legal notes
=================
| SPDX-FileCopyrightText: © 2022 ekvip automation GmbH <info@ekvip.de>
| SPDX-License-Identifier: Apache-2.0
| For details check: Apache-2.0_

.. _Apache-2.0: https://www.apache.org/licenses/LICENSE-2.0

.. </legal notes>

parameters
=================

*)

METHOD bitXIsSet
VAR_INPUT
	(* current value to check *)
	currentValue	:__XWORD;
	(* number of bit to check *)
	number			:BitNumberXWord;	
	(* message if the assertion is false *)
	message			:AssertMessage;
END_VAR
END_METHOD

(*

short summary
=================
This assertion method checks if the selected bit of current value
is unset

.. <legal notes>

legal notes
=================
| SPDX-FileCopyrightText: © 2022 ekvip automation GmbH <info@ekvip.de>
| SPDX-License-Identifier: Apache-2.0
| For details check: Apache-2.0_

.. _Apache-2.0: https://www.apache.org/licenses/LICENSE-2.0

.. </legal notes>

parameters
=================

*)

METHOD bitXIsUnset
VAR_INPUT
	(* current value to check *)
	currentValue	:__XWORD;
	(* number of bit to check *)
	number			:BitNumberXWord;	
	(* message if the assertion is false *)
	message			:AssertMessage;
END_VAR
END_METHOD

(*

short summary
=================
This assertion method checks if the least significant bit of current value
is equal to the expected value

.. <legal notes>

legal notes
=================
| SPDX-FileCopyrightText: © 2022 ekvip automation GmbH <info@ekvip.de>
| SPDX-License-Identifier: Apache-2.0
| For details check: Apache-2.0_

.. _Apache-2.0: https://www.apache.org/licenses/LICENSE-2.0

.. </legal notes>

parameters
=================

*)

METHOD lsbIsEqualTo
VAR_INPUT
	(* current value to check *)
	currentValue	:__XWORD;
	(* expected value of lsb *)
	expectedValue	:BOOL;
	(* message if the assertion is false *)
	message			:AssertMessage;
END_VAR
END_METHOD

(*

short summary
=================
This assertion method checks if the least significant bit of current value
is not equal to the unexpected value

.. <legal notes>

legal notes
=================
| SPDX-FileCopyrightText: © 2022 ekvip automation GmbH <info@ekvip.de>
| SPDX-License-Identifier: Apache-2.0
| For details check: Apache-2.0_

.. _Apache-2.0: https://www.apache.org/licenses/LICENSE-2.0

.. </legal notes>

parameters
=================

*)

METHOD lsbIsNotEqualTo
VAR_INPUT
	(* current value to check *)
	currentValue	:__XWORD;
	(* unexpected value of lsb *)
	unexpectedValue	:BOOL;
	(* message if the assertion is false *)
	message			:AssertMessage;
END_VAR
END_METHOD

(*

short summary
=================
This assertion method checks if the least significant bit of current value
is set

.. <legal notes>

legal notes
=================
| SPDX-FileCopyrightText: © 2022 ekvip automation GmbH <info@ekvip.de>
| SPDX-License-Identifier: Apache-2.0
| For details check: Apache-2.0_

.. _Apache-2.0: https://www.apache.org/licenses/LICENSE-2.0

.. </legal notes>

parameters
=================

*)

METHOD lsbIsSet
VAR_INPUT
	(* current value to check *)
	currentValue	:__XWORD;
	(* message if the assertion is false *)
	message			:AssertMessage;
END_VAR
END_METHOD

(*

short summary
=================
This assertion method checks if the least significant bit of current value
is unset

.. <legal notes>

legal notes
=================
| SPDX-FileCopyrightText: © 2022 ekvip automation GmbH <info@ekvip.de>
| SPDX-License-Identifier: Apache-2.0
| For details check: Apache-2.0_

.. _Apache-2.0: https://www.apache.org/licenses/LICENSE-2.0

.. </legal notes>

parameters
=================

*)

METHOD lsbIsUnset
VAR_INPUT
	(* current value to check *)
	currentValue	:__XWORD;
	(* message if the assertion is false *)
	message			:AssertMessage;
END_VAR
END_METHOD

(*

short summary
=================
This assertion method checks if the most significant bit of current value
is equal to the expected value

.. <legal notes>

legal notes
=================
| SPDX-FileCopyrightText: © 2022 ekvip automation GmbH <info@ekvip.de>
| SPDX-License-Identifier: Apache-2.0
| For details check: Apache-2.0_

.. _Apache-2.0: https://www.apache.org/licenses/LICENSE-2.0

.. </legal notes>

parameters
=================

*)

METHOD msbIsEqualTo
VAR_INPUT
	(* current value to check *)
	currentValue	:__XWORD;
	(* expected value of msb *)
	expectedValue	:BOOL;
	(* message if the assertion is false *)
	message			:AssertMessage;
END_VAR
END_METHOD

(*

short summary
=================
This assertion method checks if the most significant bit of current value
is not equal to the unexpected value

.. <legal notes>

legal notes
=================
| SPDX-FileCopyrightText: © 2022 ekvip automation GmbH <info@ekvip.de>
| SPDX-License-Identifier: Apache-2.0
| For details check: Apache-2.0_

.. _Apache-2.0: https://www.apache.org/licenses/LICENSE-2.0

.. </legal notes>

parameters
=================

*)

METHOD msbIsNotEqualTo
VAR_INPUT
	(* current value to check *)
	currentValue	:__XWORD;
	(* unexpected value of msb *)
	unexpectedValue	:BOOL;
	(* message if the assertion is false *)
	message			:AssertMessage;
END_VAR
END_METHOD

(*

short summary
=================
This assertion method checks if the most significant bit of current value
is set

.. <legal notes>

legal notes
=================
| SPDX-FileCopyrightText: © 2022 ekvip automation GmbH <info@ekvip.de>
| SPDX-License-Identifier: Apache-2.0
| For details check: Apache-2.0_

.. _Apache-2.0: https://www.apache.org/licenses/LICENSE-2.0

.. </legal notes>

parameters
=================

*)

METHOD msbIsSet
VAR_INPUT
	(* current value to check *)
	currentValue	:__XWORD;
	(* message if the assertion is false *)
	message			:AssertMessage;
END_VAR
END_METHOD

(*

short summary
=================
This assertion method checks if the most significant bit of current value
is unset

.. <legal notes>

legal notes
=================
| SPDX-FileCopyrightText: © 2022 ekvip automation GmbH <info@ekvip.de>
| SPDX-License-Identifier: Apache-2.0
| For details check: Apache-2.0_

.. _Apache-2.0: https://www.apache.org/licenses/LICENSE-2.0

.. </legal notes>

parameters
=================

*)

METHOD msbIsUnset
VAR_INPUT
	(* current value to check *)
	currentValue	:__XWORD;
	(* message if the assertion is false *)
	message			:AssertMessage;
END_VAR
END_METHOD

(*

short summary
=================
This assertion method checks if the result current value bitwise ``OR`` mask is equal to the expected value

.. <legal notes>

legal notes
=================
| SPDX-FileCopyrightText: © 2022 ekvip automation GmbH <info@ekvip.de>
| SPDX-License-Identifier: Apache-2.0
| For details check: Apache-2.0_

.. _Apache-2.0: https://www.apache.org/licenses/LICENSE-2.0

.. </legal notes>

parameters
=================

*)

METHOD orMaskIsEqualTo
VAR_INPUT
	(* current value to check *)
	currentValue	:__XWORD;
	(* 2nd operand for bitwise operation *)
	mask			:__XWORD;
	(* expected result after masking *)
	expectedValue	:__XWORD;
	(* message if the assertion is false *)
	message			:AssertMessage;
END_VAR
END_METHOD

(*

short summary
=================
This assertion method checks if the result current value bitwise ``OR`` mask 
is not equal to the unexpected value

.. <legal notes>

legal notes
=================
| SPDX-FileCopyrightText: © 2022 ekvip automation GmbH <info@ekvip.de>
| SPDX-License-Identifier: Apache-2.0
| For details check: Apache-2.0_

.. _Apache-2.0: https://www.apache.org/licenses/LICENSE-2.0

.. </legal notes>

parameters
=================

*)

METHOD orMaskIsNotEqualTo
VAR_INPUT
	(* current value to check *)
	currentValue	:__XWORD;
	(* 2nd operand for bitwise operation *)
	mask			:__XWORD;
	(* unexpected result after masking *)
	unexpectedValue	:__XWORD;
	(* message if the assertion is false *)
	message			:AssertMessage;
END_VAR
END_METHOD

(*

short summary
=================
This assertion method checks if the current value is equal to the expected value

.. <legal notes>

legal notes
=================
| SPDX-FileCopyrightText: © 2022 ekvip automation GmbH <info@ekvip.de>
| SPDX-License-Identifier: Apache-2.0
| For details check: Apache-2.0_

.. _Apache-2.0: https://www.apache.org/licenses/LICENSE-2.0

.. </legal notes>

parameters
=================

*)

METHOD valueIsEqualTo
VAR_INPUT
	(* current value to check *)
	currentValue	:__XWORD;
	(* expected value to compare *)
	expectedValue	:__XWORD;
	(* message if the assertion is false *)
	message			:AssertMessage;
END_VAR
END_METHOD

(*

short summary
=================
This assertion method checks if the current value is greater than the less value

.. <legal notes>

legal notes
=================
| SPDX-FileCopyrightText: © 2022 ekvip automation GmbH <info@ekvip.de>
| SPDX-License-Identifier: Apache-2.0
| For details check: Apache-2.0_

.. _Apache-2.0: https://www.apache.org/licenses/LICENSE-2.0

.. </legal notes>

parameters
=================

*)

METHOD valueIsGreaterThan
VAR_INPUT
	(* current value to check *)
	currentValue	:__XWORD;
	(* less than lower limit *)
	lessValue		:__XWORD;
	(* message if the assertion is false *)
	message			:AssertMessage;
END_VAR
END_METHOD

(*

short summary
=================
This assertion method checks if the current value is inside a limit

.. attention:: 
	limits are included: ``valueIsInRangeOf(3, 3, 3)`` is a true assertion

.. <legal notes>

legal notes
=================
| SPDX-FileCopyrightText: © 2022 ekvip automation GmbH <info@ekvip.de>
| SPDX-License-Identifier: Apache-2.0
| For details check: Apache-2.0_

.. _Apache-2.0: https://www.apache.org/licenses/LICENSE-2.0

.. </legal notes>

parameters
=================

*)

METHOD valueIsInRangeOf
VAR_INPUT
	(* lower limit for the current value *)
	lowerLimit		:__XWORD;
	(* current value to check *)
	currentValue	:__XWORD;
	(* upper limit for the current value *)
	upperLimit		:__XWORD;
	(* message if the assertion is false *)
	message			:AssertMessage;
END_VAR
END_METHOD

(*

short summary
=================
This assertion method checks if the current value is less than the greater value

.. <legal notes>

legal notes
=================
| SPDX-FileCopyrightText: © 2022 ekvip automation GmbH <info@ekvip.de>
| SPDX-License-Identifier: Apache-2.0
| For details check: Apache-2.0_

.. _Apache-2.0: https://www.apache.org/licenses/LICENSE-2.0

.. </legal notes>

parameters
=================

*)

METHOD valueIsLessThan
VAR_INPUT
	(* current value to check *)
	currentValue	:__XWORD;
	(* greater than upper limit *)
	greaterValue	:__XWORD;
	(* message if the assertion is false *)
	message			:AssertMessage;
END_VAR
END_METHOD

(*

short summary
=================
This assertion method checks if the current value is less than or equal to the maximum value

.. <legal notes>

legal notes
=================
| SPDX-FileCopyrightText: © 2022 ekvip automation GmbH <info@ekvip.de>
| SPDX-License-Identifier: Apache-2.0
| For details check: Apache-2.0_

.. _Apache-2.0: https://www.apache.org/licenses/LICENSE-2.0

.. </legal notes>

parameters
=================

*)

METHOD valueIsMax
VAR_INPUT
	(* current value to check *)
	currentValue	:__XWORD;
	(* upper limit for the current value *)
	maximumValue	:__XWORD;
	(* message if the assertion is false *)
	message			:AssertMessage;
END_VAR
END_METHOD

(*

short summary
=================
This assertion method checks if the current value is greater than or equal to the minimum value

.. <legal notes>

legal notes
=================
| SPDX-FileCopyrightText: © 2022 ekvip automation GmbH <info@ekvip.de>
| SPDX-License-Identifier: Apache-2.0
| For details check: Apache-2.0_

.. _Apache-2.0: https://www.apache.org/licenses/LICENSE-2.0

.. </legal notes>

parameters
=================

*)

METHOD valueIsMin
VAR_INPUT
	(* current value to check *)
	currentValue	:__XWORD;
	(* lower limit for the current value *)
	minimumValue	:__XWORD;
	(* message if the assertion is false *)
	message			:AssertMessage;
END_VAR
END_METHOD

(*

short summary
=================
This assertion method checks if the current value is not equal to the unexpected value

.. <legal notes>

legal notes
=================
| SPDX-FileCopyrightText: © 2022 ekvip automation GmbH <info@ekvip.de>
| SPDX-License-Identifier: Apache-2.0
| For details check: Apache-2.0_

.. _Apache-2.0: https://www.apache.org/licenses/LICENSE-2.0

.. </legal notes>

parameters
=================

*)

METHOD valueIsNotEqualTo
VAR_INPUT
	(* current value to check *)
	currentValue	:__XWORD;
	(* unexpected value to compare *)
	unexpectedValue	:__XWORD;
	(* message if the assertion is false *)
	message			:AssertMessage;
END_VAR
END_METHOD

(*

short summary
=================
This assertion method checks if the result current value bitwise ``XOR`` mask is equal to the expected value

.. <legal notes>

legal notes
=================
| SPDX-FileCopyrightText: © 2022 ekvip automation GmbH <info@ekvip.de>
| SPDX-License-Identifier: Apache-2.0
| For details check: Apache-2.0_

.. _Apache-2.0: https://www.apache.org/licenses/LICENSE-2.0

.. </legal notes>

parameters
=================

*)

METHOD xorMaskIsEqualTo
VAR_INPUT
	(* current value to check *)
	currentValue	:__XWORD;
	(* 2nd operand for bitwise operation *)
	mask			:__XWORD;
	(* expected result after masking *)
	expectedValue	:__XWORD;
	(* message if the assertion is false *)
	message			:AssertMessage;
END_VAR
END_METHOD

(*

short summary
=================
This assertion method checks if the result current value bitwise ``XOR`` mask 
is not equal to the unexpected value

.. <legal notes>

legal notes
=================
| SPDX-FileCopyrightText: © 2022 ekvip automation GmbH <info@ekvip.de>
| SPDX-License-Identifier: Apache-2.0
| For details check: Apache-2.0_

.. _Apache-2.0: https://www.apache.org/licenses/LICENSE-2.0

.. </legal notes>

parameters
=================

*)

METHOD xorMaskIsNotEqualTo
VAR_INPUT
	(* current value to check *)
	currentValue	:__XWORD;
	(* 2nd operand for bitwise operation *)
	mask			:__XWORD;
	(* unexpected result after masking *)
	unexpectedValue	:__XWORD;
	(* message if the assertion is false *)
	message			:AssertMessage;
END_VAR
END_METHOD

END_INTERFACE

// ---- Assertor/Assertions/BooleanAssertion/interfaces/IBooleanAssertion.TcIO
(*

short summary
=================
This interface provides assert statements for booleans 

.. <legal notes>

legal notes
=================
| SPDX-FileCopyrightText: © 2022 ekvip automation GmbH <info@ekvip.de>
| SPDX-License-Identifier: Apache-2.0
| For details check: Apache-2.0_

.. _Apache-2.0: https://www.apache.org/licenses/LICENSE-2.0

.. </legal notes>

methods
==================

*)

INTERFACE IBooleanAssertion EXTENDS __SYSTEM.IQueryInterface

(*

short summary
=================
This assertion method checks if the current value is equal to the expected value

.. <legal notes>

legal notes
=================
| SPDX-FileCopyrightText: © 2022 ekvip automation GmbH <info@ekvip.de>
| SPDX-License-Identifier: Apache-2.0
| For details check: Apache-2.0_

.. _Apache-2.0: https://www.apache.org/licenses/LICENSE-2.0

.. </legal notes>

parameters
=================

*)

METHOD valueIsEqualTo
VAR_INPUT
	(* current value to check *)
	currentValue	:BOOL;
	(* expected value to compare *)
	expectedValue	:BOOL;
	(* message if the assertion is false *)
	message			:AssertMessage;
END_VAR
END_METHOD

(*

short summary
=================
This assertion method checks if the current value is ``FALSE``

.. <legal notes>

legal notes
=================
| SPDX-FileCopyrightText: © 2022 ekvip automation GmbH <info@ekvip.de>
| SPDX-License-Identifier: Apache-2.0
| For details check: Apache-2.0_

.. _Apache-2.0: https://www.apache.org/licenses/LICENSE-2.0

.. </legal notes>

parameters
=================

*)

METHOD valueIsFalse
VAR_INPUT
	(* current value to check *)
	currentValue	:BOOL;
	(* message if the assertion is false *)
	message			:AssertMessage;
END_VAR
END_METHOD

(*

short summary
=================
This assertion method checks if the current value is not equal to the unexpected value

.. <legal notes>

legal notes
=================
| SPDX-FileCopyrightText: © 2022 ekvip automation GmbH <info@ekvip.de>
| SPDX-License-Identifier: Apache-2.0
| For details check: Apache-2.0_

.. _Apache-2.0: https://www.apache.org/licenses/LICENSE-2.0

.. </legal notes>

parameters
=================

*)

METHOD valueIsNotEqualTo
VAR_INPUT
	(* current value to check *)
	currentValue	:BOOL;
	(* unexpected value to compare *)
	unexpectedValue	:BOOL;
	(* message if the assertion is false *)
	message			:AssertMessage;
END_VAR
END_METHOD

(*

short summary
=================
This assertion method checks if the current value is ``TRUE``

.. <legal notes>

legal notes
=================
| SPDX-FileCopyrightText: © 2022 ekvip automation GmbH <info@ekvip.de>
| SPDX-License-Identifier: Apache-2.0
| For details check: Apache-2.0_

.. _Apache-2.0: https://www.apache.org/licenses/LICENSE-2.0

.. </legal notes>

parameters
=================

*)

METHOD valueIsTrue
VAR_INPUT
	(* current value to check *)
	currentValue	:BOOL;
	(* message if the assertion is false *)
	message			:AssertMessage;
END_VAR
END_METHOD

END_INTERFACE

// ---- Assertor/Assertions/DateAndTimeAssertions/32Bit/Date/interfaces/I32BitDateAssertions.TcIO
(*

short summary
=================
This interface provides assert statements for 32 bit ``DATE``  

.. <legal notes>

legal notes
=================
| SPDX-FileCopyrightText: © 2022 ekvip automation GmbH <info@ekvip.de>
| SPDX-License-Identifier: Apache-2.0
| For details check: Apache-2.0_

.. _Apache-2.0: https://www.apache.org/licenses/LICENSE-2.0

.. </legal notes>

methods
==================

*)

INTERFACE I32BitDateAssertions EXTENDS __SYSTEM.IQueryInterface

(*

short summary
=================
This assertion method checks if the current value is equal to the expected value

.. <legal notes>

legal notes
=================
| SPDX-FileCopyrightText: © 2022 ekvip automation GmbH <info@ekvip.de>
| SPDX-License-Identifier: Apache-2.0
| For details check: Apache-2.0_

.. _Apache-2.0: https://www.apache.org/licenses/LICENSE-2.0

.. </legal notes>

parameters
=================

*)

METHOD valueIsEqualTo
VAR_INPUT
	(* current value to check *)
	currentValue	:DATE;
	(* expected value to compare *)
	expectedValue	:DATE;
	(* message if the assertion is false *)
	message			:AssertMessage;
END_VAR
END_METHOD

(*

short summary
=================
This assertion method checks if the current value is greater than the less value

.. <legal notes>

legal notes
=================
| SPDX-FileCopyrightText: © 2022 ekvip automation GmbH <info@ekvip.de>
| SPDX-License-Identifier: Apache-2.0
| For details check: Apache-2.0_

.. _Apache-2.0: https://www.apache.org/licenses/LICENSE-2.0

.. </legal notes>

parameters
=================

*)

METHOD valueIsGreaterThan
VAR_INPUT
	(* current value to check *)
	currentValue	:DATE;
	(* less than lower limit *)
	lessValue		:DATE;
	(* message if the assertion is false *)
	message			:AssertMessage;
END_VAR
END_METHOD

(*

short summary
=================
This assertion method checks if the current value is inside a limit

.. attention:: 
	limits are included: ``valueIsInRangeOf(date#1970-01-01, date#1970-01-01, date#1970-01-01)``
	is a true assertion

.. <legal notes>

legal notes
=================
| SPDX-FileCopyrightText: © 2022 ekvip automation GmbH <info@ekvip.de>
| SPDX-License-Identifier: Apache-2.0
| For details check: Apache-2.0_

.. _Apache-2.0: https://www.apache.org/licenses/LICENSE-2.0

.. </legal notes>

parameters
=================

*)

METHOD valueIsInRangeOf
VAR_INPUT
	(* lower limit for the current value *)
	lowerLimit		:DATE;
	(* current value to check *)
	currentValue	:DATE;
	(* upper limit for the current value *)
	upperLimit		:DATE;
	(* message if the assertion is false *)
	message			:AssertMessage;
END_VAR
END_METHOD

(*

short summary
=================
This assertion method checks if the current value is less than the greater value

.. <legal notes>

legal notes
=================
| SPDX-FileCopyrightText: © 2022 ekvip automation GmbH <info@ekvip.de>
| SPDX-License-Identifier: Apache-2.0
| For details check: Apache-2.0_

.. _Apache-2.0: https://www.apache.org/licenses/LICENSE-2.0

.. </legal notes>

parameters
=================

*)

METHOD valueIsLessThan
VAR_INPUT
	(* current value to check *)
	currentValue	:DATE;
	(* greater than upper limit *)
	greaterValue	:DATE;
	(* message if the assertion is false *)
	message			:AssertMessage;
END_VAR
END_METHOD

(*

short summary
=================
This assertion method checks if the current value is less than or equal to the maximum value

.. <legal notes>

legal notes
=================
| SPDX-FileCopyrightText: © 2022 ekvip automation GmbH <info@ekvip.de>
| SPDX-License-Identifier: Apache-2.0
| For details check: Apache-2.0_

.. _Apache-2.0: https://www.apache.org/licenses/LICENSE-2.0

.. </legal notes>

parameters
=================

*)

METHOD valueIsMax
VAR_INPUT
	(* current value to check *)
	currentValue	:DATE;
	(* upper limit for the current value *)
	maximumValue	:DATE;
	(* message if the assertion is false *)
	message			:AssertMessage;
END_VAR
END_METHOD

(*

short summary
=================
This assertion method checks if the current value is greater than or equal to the minimum value

.. <legal notes>

legal notes
=================
| SPDX-FileCopyrightText: © 2022 ekvip automation GmbH <info@ekvip.de>
| SPDX-License-Identifier: Apache-2.0
| For details check: Apache-2.0_

.. _Apache-2.0: https://www.apache.org/licenses/LICENSE-2.0

.. </legal notes>

parameters
=================

*)

METHOD valueIsMin
VAR_INPUT
	(* current value to check *)
	currentValue	:DATE;
	(* lower limit for the current value *)
	minimumValue	:DATE;
	(* message if the assertion is false *)
	message			:AssertMessage;
END_VAR
END_METHOD

(*

short summary
=================
This assertion method checks if the current value is not equal to the unexpected value

.. <legal notes>

legal notes
=================
| SPDX-FileCopyrightText: © 2022 ekvip automation GmbH <info@ekvip.de>
| SPDX-License-Identifier: Apache-2.0
| For details check: Apache-2.0_

.. _Apache-2.0: https://www.apache.org/licenses/LICENSE-2.0

.. </legal notes>

parameters
=================

*)

METHOD valueIsNotEqualTo
VAR_INPUT
	(* current value to check *)
	currentValue	:DATE;
	(* unexpected value to compare *)
	unexpectedValue	:DATE;
	(* message if the assertion is false *)
	message			:AssertMessage;
END_VAR
END_METHOD

END_INTERFACE

// ---- Assertor/Assertions/DateAndTimeAssertions/32Bit/DT/interfaces/I32BitDtAssertions.TcIO
(*

short summary
=================
This interface provides assert statements for 32 bit date and time ``DT``  

.. <legal notes>

legal notes
=================
| SPDX-FileCopyrightText: © 2022 ekvip automation GmbH <info@ekvip.de>
| SPDX-License-Identifier: Apache-2.0
| For details check: Apache-2.0_

.. _Apache-2.0: https://www.apache.org/licenses/LICENSE-2.0

.. </legal notes>

methods
==================

*)

INTERFACE I32BitDtAssertions EXTENDS __SYSTEM.IQueryInterface

(*

short summary
=================
This assertion method checks if the current value is equal to the expected value

.. <legal notes>

legal notes
=================
| SPDX-FileCopyrightText: © 2022 ekvip automation GmbH <info@ekvip.de>
| SPDX-License-Identifier: Apache-2.0
| For details check: Apache-2.0_

.. _Apache-2.0: https://www.apache.org/licenses/LICENSE-2.0

.. </legal notes>

parameters
=================

*)

METHOD valueIsEqualTo
VAR_INPUT
	(* current value to check *)
	currentValue	:DT;
	(* expected value to compare *)
	expectedValue	:DT;
	(* message if the assertion is false *)
	message			:AssertMessage;
END_VAR
END_METHOD

(*

short summary
=================
This assertion method checks if the current value is greater than the less value

.. <legal notes>

legal notes
=================
| SPDX-FileCopyrightText: © 2022 ekvip automation GmbH <info@ekvip.de>
| SPDX-License-Identifier: Apache-2.0
| For details check: Apache-2.0_

.. _Apache-2.0: https://www.apache.org/licenses/LICENSE-2.0

.. </legal notes>

parameters
=================

*)

METHOD valueIsGreaterThan
VAR_INPUT
	(* current value to check *)
	currentValue	:DT;
	(* less than lower limit *)
	lessValue		:DT;
	(* message if the assertion is false *)
	message			:AssertMessage;
END_VAR
END_METHOD

(*

short summary
=================
This assertion method checks if the current value is inside a limit

.. attention:: 
	limits are included: ``valueIsInRangeOf(dt#1970-01-01-0:0:0, dt#1970-01-01-0:0:0, dt#1970-01-01-0:0:0)``
	is a true assertion

.. <legal notes>

legal notes
=================
| SPDX-FileCopyrightText: © 2022 ekvip automation GmbH <info@ekvip.de>
| SPDX-License-Identifier: Apache-2.0
| For details check: Apache-2.0_

.. _Apache-2.0: https://www.apache.org/licenses/LICENSE-2.0

.. </legal notes>

parameters
=================

*)

METHOD valueIsInRangeOf
VAR_INPUT
	(* lower limit for the current value *)
	lowerLimit		:DT;
	(* current value to check *)
	currentValue	:DT;
	(* upper limit for the current value *)
	upperLimit		:DT;
	(* message if the assertion is false *)
	message			:AssertMessage;
END_VAR
END_METHOD

(*

short summary
=================
This assertion method checks if the current value is less than the greater value

.. <legal notes>

legal notes
=================
| SPDX-FileCopyrightText: © 2022 ekvip automation GmbH <info@ekvip.de>
| SPDX-License-Identifier: Apache-2.0
| For details check: Apache-2.0_

.. _Apache-2.0: https://www.apache.org/licenses/LICENSE-2.0

.. </legal notes>

parameters
=================

*)

METHOD valueIsLessThan
VAR_INPUT
	(* current value to check *)
	currentValue	:DT;
	(* greater than upper limit *)
	greaterValue	:DT;
	(* message if the assertion is false *)
	message			:AssertMessage;
END_VAR
END_METHOD

(*

short summary
=================
This assertion method checks if the current value is less than or equal to the maximum value

.. <legal notes>

legal notes
=================
| SPDX-FileCopyrightText: © 2022 ekvip automation GmbH <info@ekvip.de>
| SPDX-License-Identifier: Apache-2.0
| For details check: Apache-2.0_

.. _Apache-2.0: https://www.apache.org/licenses/LICENSE-2.0

.. </legal notes>

parameters
=================

*)

METHOD valueIsMax
VAR_INPUT
	(* current value to check *)
	currentValue	:DT;
	(* upper limit for the current value *)
	maximumValue	:DT;
	(* message if the assertion is false *)
	message			:AssertMessage;
END_VAR
END_METHOD

(*

short summary
=================
This assertion method checks if the current value is greater than or equal to the minimum value

.. <legal notes>

legal notes
=================
| SPDX-FileCopyrightText: © 2022 ekvip automation GmbH <info@ekvip.de>
| SPDX-License-Identifier: Apache-2.0
| For details check: Apache-2.0_

.. _Apache-2.0: https://www.apache.org/licenses/LICENSE-2.0

.. </legal notes>

parameters
=================

*)

METHOD valueIsMin
VAR_INPUT
	(* current value to check *)
	currentValue	:DT;
	(* lower limit for the current value *)
	minimumValue	:DT;
	(* message if the assertion is false *)
	message			:AssertMessage;
END_VAR
END_METHOD

(*

short summary
=================
This assertion method checks if the current value is not equal to the unexpected value

.. <legal notes>

legal notes
=================
| SPDX-FileCopyrightText: © 2022 ekvip automation GmbH <info@ekvip.de>
| SPDX-License-Identifier: Apache-2.0
| For details check: Apache-2.0_

.. _Apache-2.0: https://www.apache.org/licenses/LICENSE-2.0

.. </legal notes>

parameters
=================

*)

METHOD valueIsNotEqualTo
VAR_INPUT
	(* current value to check *)
	currentValue	:DT;
	(* unexpected value to compare *)
	unexpectedValue	:DT;
	(* message if the assertion is false *)
	message			:AssertMessage;
END_VAR
END_METHOD

END_INTERFACE

// ---- Assertor/Assertions/DateAndTimeAssertions/32Bit/interfaces/ISimpleDateAndTimeAssertions.TcIO
(*

short summary
=================
| This interface provides assert statements for date and time types with 32 bit length
| For date and time (``DT``) use :ref:`ISimpleDateAndTimeAssertions.dateAndTime`
| For date (``DATE``) use  :ref:`ISimpleDateAndTimeAssertions.dateOnly`
| For time of day (``TOD``) use  :ref:`ISimpleDateAndTimeAssertions.timeOfDay`

.. <legal notes>

legal notes
=================
| SPDX-FileCopyrightText: © 2022 ekvip automation GmbH <info@ekvip.de>
| SPDX-License-Identifier: Apache-2.0
| For details check: Apache-2.0_

.. _Apache-2.0: https://www.apache.org/licenses/LICENSE-2.0

.. </legal notes>

methods
==================

*)

INTERFACE ISimpleDateAndTimeAssertions EXTENDS __SYSTEM.IQueryInterface

(*

short summary
=================
Returns the interface :ref:`I32BitDtAssertions` with assert statements for 32 bit date and time ``DT``

.. <legal notes>

legal notes
=================
| SPDX-FileCopyrightText: © 2022 ekvip automation GmbH <info@ekvip.de>
| SPDX-License-Identifier: Apache-2.0
| For details check: Apache-2.0_

.. _Apache-2.0: https://www.apache.org/licenses/LICENSE-2.0

.. </legal notes>

*)

PROPERTY dateAndTime :I32BitDtAssertions
GET
END_GET
END_PROPERTY

(*

short summary
=================
Returns the interface :ref:`I32BitDateAssertions` with assert statements for 32 bit date ``DATE``

.. <legal notes>

legal notes
=================
| SPDX-FileCopyrightText: © 2022 ekvip automation GmbH <info@ekvip.de>
| SPDX-License-Identifier: Apache-2.0
| For details check: Apache-2.0_

.. _Apache-2.0: https://www.apache.org/licenses/LICENSE-2.0

.. </legal notes>

*)

PROPERTY dateOnly :I32BitDateAssertions
GET
END_GET
END_PROPERTY

(*

short summary
=================
Returns the interface :ref:`I32BitTodAssertions` with assert statements for 32 bit time of day ``TOD``

.. <legal notes>

legal notes
=================
| SPDX-FileCopyrightText: © 2022 ekvip automation GmbH <info@ekvip.de>
| SPDX-License-Identifier: Apache-2.0
| For details check: Apache-2.0_

.. _Apache-2.0: https://www.apache.org/licenses/LICENSE-2.0

.. </legal notes>

*)

PROPERTY timeOfDay :I32BitTodAssertions
GET
END_GET
END_PROPERTY

END_INTERFACE

// ---- Assertor/Assertions/DateAndTimeAssertions/32Bit/TOD/interfaces/I32BitTodAssertions.TcIO
(*

short summary
=================
This interface provides assert statements for 32 bit time of day ``TOD``  

.. <legal notes>

legal notes
=================
| SPDX-FileCopyrightText: © 2022 ekvip automation GmbH <info@ekvip.de>
| SPDX-License-Identifier: Apache-2.0
| For details check: Apache-2.0_

.. _Apache-2.0: https://www.apache.org/licenses/LICENSE-2.0

.. </legal notes>

methods
==================

*)

INTERFACE I32BitTodAssertions EXTENDS __SYSTEM.IQueryInterface

(*

short summary
=================
This assertion method checks if the current value is equal to the expected value

.. <legal notes>

legal notes
=================
| SPDX-FileCopyrightText: © 2022 ekvip automation GmbH <info@ekvip.de>
| SPDX-License-Identifier: Apache-2.0
| For details check: Apache-2.0_

.. _Apache-2.0: https://www.apache.org/licenses/LICENSE-2.0

.. </legal notes>

parameters
=================

*)

METHOD valueIsEqualTo
VAR_INPUT
	(* current value to check *)
	currentValue	:TOD;
	(* expected value to compare *)
	expectedValue	:TOD;
	(* message if the assertion is false *)
	message			:AssertMessage;
END_VAR
END_METHOD

(*

short summary
=================
This assertion method checks if the current value is greater than the less value

.. <legal notes>

legal notes
=================
| SPDX-FileCopyrightText: © 2022 ekvip automation GmbH <info@ekvip.de>
| SPDX-License-Identifier: Apache-2.0
| For details check: Apache-2.0_

.. _Apache-2.0: https://www.apache.org/licenses/LICENSE-2.0

.. </legal notes>

parameters
=================

*)

METHOD valueIsGreaterThan
VAR_INPUT
	(* current value to check *)
	currentValue	:TOD;
	(* less than lower limit *)
	lessValue		:TOD;
	(* message if the assertion is false *)
	message			:AssertMessage;
END_VAR
END_METHOD

(*

short summary
=================
This assertion method checks if the current value is inside a limit

.. attention:: 
	limits are included: ``valueIsInRangeOf(tod#3:0:0, tod#3:0:0, tod#3:0:0)`` is a true assertion

.. <legal notes>

legal notes
=================
| SPDX-FileCopyrightText: © 2022 ekvip automation GmbH <info@ekvip.de>
| SPDX-License-Identifier: Apache-2.0
| For details check: Apache-2.0_

.. _Apache-2.0: https://www.apache.org/licenses/LICENSE-2.0

.. </legal notes>

parameters
=================

*)

METHOD valueIsInRangeOf
VAR_INPUT
	(* lower limit for the current value *)
	lowerLimit		:TOD;
	(* current value to check *)
	currentValue	:TOD;
	(* upper limit for the current value *)
	upperLimit		:TOD;
	(* message if the assertion is false *)
	message			:AssertMessage;
END_VAR
END_METHOD

(*

short summary
=================
This assertion method checks if the current value is less than the greater value

.. <legal notes>

legal notes
=================
| SPDX-FileCopyrightText: © 2022 ekvip automation GmbH <info@ekvip.de>
| SPDX-License-Identifier: Apache-2.0
| For details check: Apache-2.0_

.. _Apache-2.0: https://www.apache.org/licenses/LICENSE-2.0

.. </legal notes>

parameters
=================

*)

METHOD valueIsLessThan
VAR_INPUT
	(* current value to check *)
	currentValue	:TOD;
	(* greater than upper limit *)
	greaterValue	:TOD;
	(* message if the assertion is false *)
	message			:AssertMessage;
END_VAR
END_METHOD

(*

short summary
=================
This assertion method checks if the current value is less than or equal to the maximum value

.. <legal notes>

legal notes
=================
| SPDX-FileCopyrightText: © 2022 ekvip automation GmbH <info@ekvip.de>
| SPDX-License-Identifier: Apache-2.0
| For details check: Apache-2.0_

.. _Apache-2.0: https://www.apache.org/licenses/LICENSE-2.0

.. </legal notes>

parameters
=================

*)

METHOD valueIsMax
VAR_INPUT
	(* current value to check *)
	currentValue	:TOD;
	(* upper limit for the current value *)
	maximumValue	:TOD;
	(* message if the assertion is false *)
	message			:AssertMessage;
END_VAR
END_METHOD

(*

short summary
=================
This assertion method checks if the current value is greater than or equal to the minimum value

.. <legal notes>

legal notes
=================
| SPDX-FileCopyrightText: © 2022 ekvip automation GmbH <info@ekvip.de>
| SPDX-License-Identifier: Apache-2.0
| For details check: Apache-2.0_

.. _Apache-2.0: https://www.apache.org/licenses/LICENSE-2.0

.. </legal notes>

parameters
=================

*)

METHOD valueIsMin
VAR_INPUT
	(* current value to check *)
	currentValue	:TOD;
	(* lower limit for the current value *)
	minimumValue	:TOD;
	(* message if the assertion is false *)
	message			:AssertMessage;
END_VAR
END_METHOD

(*

short summary
=================
This assertion method checks if the current value is not equal to the unexpected value

.. <legal notes>

legal notes
=================
| SPDX-FileCopyrightText: © 2022 ekvip automation GmbH <info@ekvip.de>
| SPDX-License-Identifier: Apache-2.0
| For details check: Apache-2.0_

.. _Apache-2.0: https://www.apache.org/licenses/LICENSE-2.0

.. </legal notes>

parameters
=================

*)

METHOD valueIsNotEqualTo
VAR_INPUT
	(* current value to check *)
	currentValue	:TOD;
	(* unexpected value to compare *)
	unexpectedValue	:TOD;
	(* message if the assertion is false *)
	message			:AssertMessage;
END_VAR
END_METHOD

END_INTERFACE

// ---- Assertor/Assertions/DateAndTimeAssertions/64Bit/LDate/interfaces/I64BitDateAssertions.TcIO
(*

short summary
=================
This interface provides assert statements for 32 bit ``DATE``  

.. <legal notes>

legal notes
=================
| SPDX-FileCopyrightText: © 2022 ekvip automation GmbH <info@ekvip.de>
| SPDX-License-Identifier: Apache-2.0
| For details check: Apache-2.0_

.. _Apache-2.0: https://www.apache.org/licenses/LICENSE-2.0

.. </legal notes>

methods
==================

*)

INTERFACE I64BitDateAssertions EXTENDS __SYSTEM.IQueryInterface

(*

short summary
=================
This assertion method checks if the current value is equal to the expected value

.. <legal notes>

legal notes
=================
| SPDX-FileCopyrightText: © 2022 ekvip automation GmbH <info@ekvip.de>
| SPDX-License-Identifier: Apache-2.0
| For details check: Apache-2.0_

.. _Apache-2.0: https://www.apache.org/licenses/LICENSE-2.0

.. </legal notes>

parameters
=================

*)

METHOD valueIsEqualTo
VAR_INPUT
	(* current value to check *)
	currentValue	:LDATE;
	(* expected value to compare *)
	expectedValue	:LDATE;
	(* message if the assertion is false *)
	message			:AssertMessage;
END_VAR
END_METHOD

(*

short summary
=================
This assertion method checks if the current value is greater than the less value

.. <legal notes>

legal notes
=================
| SPDX-FileCopyrightText: © 2022 ekvip automation GmbH <info@ekvip.de>
| SPDX-License-Identifier: Apache-2.0
| For details check: Apache-2.0_

.. _Apache-2.0: https://www.apache.org/licenses/LICENSE-2.0

.. </legal notes>

parameters
=================

*)

METHOD valueIsGreaterThan
VAR_INPUT
	(* current value to check *)
	currentValue	:LDATE;
	(* less than lower limit *)
	lessValue		:LDATE;
	(* message if the assertion is false *)
	message			:AssertMessage;
END_VAR
END_METHOD

(*

short summary
=================
This assertion method checks if the current value is inside a limit

.. attention:: 
	limits are included: ``valueIsInRangeOf(ldate#1970-01-01, ldate#1970-01-01, ldate#1970-01-01)``
	is a true assertion

.. <legal notes>

legal notes
=================
| SPDX-FileCopyrightText: © 2022 ekvip automation GmbH <info@ekvip.de>
| SPDX-License-Identifier: Apache-2.0
| For details check: Apache-2.0_

.. _Apache-2.0: https://www.apache.org/licenses/LICENSE-2.0

.. </legal notes>

parameters
=================

*)

METHOD valueIsInRangeOf
VAR_INPUT
	(* lower limit for the current value *)
	lowerLimit		:LDATE;
	(* current value to check *)
	currentValue	:LDATE;
	(* upper limit for the current value *)
	upperLimit		:LDATE;
	(* message if the assertion is false *)
	message			:AssertMessage;
END_VAR
END_METHOD

(*

short summary
=================
This assertion method checks if the current value is less than the greater value

.. <legal notes>

legal notes
=================
| SPDX-FileCopyrightText: © 2022 ekvip automation GmbH <info@ekvip.de>
| SPDX-License-Identifier: Apache-2.0
| For details check: Apache-2.0_

.. _Apache-2.0: https://www.apache.org/licenses/LICENSE-2.0

.. </legal notes>

parameters
=================

*)

METHOD valueIsLessThan
VAR_INPUT
	(* current value to check *)
	currentValue	:LDATE;
	(* greater than upper limit *)
	greaterValue	:LDATE;
	(* message if the assertion is false *)
	message			:AssertMessage;
END_VAR
END_METHOD

(*

short summary
=================
This assertion method checks if the current value is less than or equal to the maximum value

.. <legal notes>

legal notes
=================
| SPDX-FileCopyrightText: © 2022 ekvip automation GmbH <info@ekvip.de>
| SPDX-License-Identifier: Apache-2.0
| For details check: Apache-2.0_

.. _Apache-2.0: https://www.apache.org/licenses/LICENSE-2.0

.. </legal notes>

parameters
=================

*)

METHOD valueIsMax
VAR_INPUT
	(* current value to check *)
	currentValue	:LDATE;
	(* upper limit for the current value *)
	maximumValue	:LDATE;
	(* message if the assertion is false *)
	message			:AssertMessage;
END_VAR
END_METHOD

(*

short summary
=================
This assertion method checks if the current value is greater than or equal to the minimum value

.. <legal notes>

legal notes
=================
| SPDX-FileCopyrightText: © 2022 ekvip automation GmbH <info@ekvip.de>
| SPDX-License-Identifier: Apache-2.0
| For details check: Apache-2.0_

.. _Apache-2.0: https://www.apache.org/licenses/LICENSE-2.0

.. </legal notes>

parameters
=================

*)

METHOD valueIsMin
VAR_INPUT
	(* current value to check *)
	currentValue	:LDATE;
	(* lower limit for the current value *)
	minimumValue	:LDATE;
	(* message if the assertion is false *)
	message			:AssertMessage;
END_VAR
END_METHOD

(*

short summary
=================
This assertion method checks if the current value is not equal to the unexpected value

.. <legal notes>

legal notes
=================
| SPDX-FileCopyrightText: © 2022 ekvip automation GmbH <info@ekvip.de>
| SPDX-License-Identifier: Apache-2.0
| For details check: Apache-2.0_

.. _Apache-2.0: https://www.apache.org/licenses/LICENSE-2.0

.. </legal notes>

parameters
=================

*)

METHOD valueIsNotEqualTo
VAR_INPUT
	(* current value to check *)
	currentValue	:LDATE;
	(* unexpected value to compare *)
	unexpectedValue	:LDATE;
	(* message if the assertion is false *)
	message			:AssertMessage;
END_VAR
END_METHOD

END_INTERFACE

// ---- Assertor/Assertions/DateAndTimeAssertions/64Bit/LDT/interfaces/I64BitDtAssertions.TcIO
(*

short summary
=================
This interface provides assert statements for 64 bit date and time ``LDT``  

.. <legal notes>

legal notes
=================
| SPDX-FileCopyrightText: © 2022 ekvip automation GmbH <info@ekvip.de>
| SPDX-License-Identifier: Apache-2.0
| For details check: Apache-2.0_

.. _Apache-2.0: https://www.apache.org/licenses/LICENSE-2.0

.. </legal notes>

methods
==================

*)

INTERFACE I64BitDtAssertions EXTENDS __SYSTEM.IQueryInterface

(*

short summary
=================
This assertion method checks if the current value is equal to the expected value

.. <legal notes>

legal notes
=================
| SPDX-FileCopyrightText: © 2022 ekvip automation GmbH <info@ekvip.de>
| SPDX-License-Identifier: Apache-2.0
| For details check: Apache-2.0_

.. _Apache-2.0: https://www.apache.org/licenses/LICENSE-2.0

.. </legal notes>

parameters
=================

*)

METHOD valueIsEqualTo
VAR_INPUT
	(* current value to check *)
	currentValue	:LDT;
	(* expected value to compare *)
	expectedValue	:LDT;
	(* message if the assertion is false *)
	message			:AssertMessage;
END_VAR
END_METHOD

(*

short summary
=================
This assertion method checks if the current value is greater than the less value

.. <legal notes>

legal notes
=================
| SPDX-FileCopyrightText: © 2022 ekvip automation GmbH <info@ekvip.de>
| SPDX-License-Identifier: Apache-2.0
| For details check: Apache-2.0_

.. _Apache-2.0: https://www.apache.org/licenses/LICENSE-2.0

.. </legal notes>

parameters
=================

*)

METHOD valueIsGreaterThan
VAR_INPUT
	(* current value to check *)
	currentValue	:LDT;
	(* less than lower limit *)
	lessValue		:LDT;
	(* message if the assertion is false *)
	message			:AssertMessage;
END_VAR
END_METHOD

(*

short summary
=================
This assertion method checks if the current value is inside a limit

.. attention:: 
	limits are included: ``valueIsInRangeOf(ldt#1970-01-01-0:0:0, ldt#1970-01-01-0:0:0, ldt#1970-01-01-0:0:0)``
	is a true assertion

.. <legal notes>

legal notes
=================
| SPDX-FileCopyrightText: © 2022 ekvip automation GmbH <info@ekvip.de>
| SPDX-License-Identifier: Apache-2.0
| For details check: Apache-2.0_

.. _Apache-2.0: https://www.apache.org/licenses/LICENSE-2.0

.. </legal notes>

parameters
=================

*)

METHOD valueIsInRangeOf
VAR_INPUT
	(* lower limit for the current value *)
	lowerLimit		:LDT;
	(* current value to check *)
	currentValue	:LDT;
	(* upper limit for the current value *)
	upperLimit		:LDT;
	(* message if the assertion is false *)
	message			:AssertMessage;
END_VAR
END_METHOD

(*

short summary
=================
This assertion method checks if the current value is less than the greater value

.. <legal notes>

legal notes
=================
| SPDX-FileCopyrightText: © 2022 ekvip automation GmbH <info@ekvip.de>
| SPDX-License-Identifier: Apache-2.0
| For details check: Apache-2.0_

.. _Apache-2.0: https://www.apache.org/licenses/LICENSE-2.0

.. </legal notes>

parameters
=================

*)

METHOD valueIsLessThan
VAR_INPUT
	(* current value to check *)
	currentValue	:LDT;
	(* greater than upper limit *)
	greaterValue	:LDT;
	(* message if the assertion is false *)
	message			:AssertMessage;
END_VAR
END_METHOD

(*

short summary
=================
This assertion method checks if the current value is less than or equal to the maximum value

.. <legal notes>

legal notes
=================
| SPDX-FileCopyrightText: © 2022 ekvip automation GmbH <info@ekvip.de>
| SPDX-License-Identifier: Apache-2.0
| For details check: Apache-2.0_

.. _Apache-2.0: https://www.apache.org/licenses/LICENSE-2.0

.. </legal notes>

parameters
=================

*)

METHOD valueIsMax
VAR_INPUT
	(* current value to check *)
	currentValue	:LDT;
	(* upper limit for the current value *)
	maximumValue	:LDT;
	(* message if the assertion is false *)
	message			:AssertMessage;
END_VAR
END_METHOD

(*

short summary
=================
This assertion method checks if the current value is greater than or equal to the minimum value

.. <legal notes>

legal notes
=================
| SPDX-FileCopyrightText: © 2022 ekvip automation GmbH <info@ekvip.de>
| SPDX-License-Identifier: Apache-2.0
| For details check: Apache-2.0_

.. _Apache-2.0: https://www.apache.org/licenses/LICENSE-2.0

.. </legal notes>

parameters
=================

*)

METHOD valueIsMin
VAR_INPUT
	(* current value to check *)
	currentValue	:LDT;
	(* lower limit for the current value *)
	minimumValue	:LDT;
	(* message if the assertion is false *)
	message			:AssertMessage;
END_VAR
END_METHOD

(*

short summary
=================
This assertion method checks if the current value is not equal to the unexpected value

.. <legal notes>

legal notes
=================
| SPDX-FileCopyrightText: © 2022 ekvip automation GmbH <info@ekvip.de>
| SPDX-License-Identifier: Apache-2.0
| For details check: Apache-2.0_

.. _Apache-2.0: https://www.apache.org/licenses/LICENSE-2.0

.. </legal notes>

parameters
=================

*)

METHOD valueIsNotEqualTo
VAR_INPUT
	(* current value to check *)
	currentValue	:LDT;
	(* unexpected value to compare *)
	unexpectedValue	:LDT;
	(* message if the assertion is false *)
	message			:AssertMessage;
END_VAR
END_METHOD

END_INTERFACE

// ---- Assertor/Assertions/DateAndTimeAssertions/64Bit/interfaces/ILongDateAndTimeAssertions.TcIO
(*

short summary
=================
| This interface provides assert statements for date and time types with 64 bit length
| For date and time (``LDT``) use :ref:`ISimpleDateAndTimeAssertions.dateAndTime`
| For date (``LDATE``) use  :ref:`ISimpleDateAndTimeAssertions.dateOnly`
| For time of day (``LTOD``) use  :ref:`ISimpleDateAndTimeAssertions.timeOfDay`

.. <legal notes>

legal notes
=================
| SPDX-FileCopyrightText: © 2022 ekvip automation GmbH <info@ekvip.de>
| SPDX-License-Identifier: Apache-2.0
| For details check: Apache-2.0_

.. _Apache-2.0: https://www.apache.org/licenses/LICENSE-2.0

.. </legal notes>

methods
==================

*)

INTERFACE ILongDateAndTimeAssertions EXTENDS __SYSTEM.IQueryInterface

(*

short summary
=================
Returns the interface :ref:`I64BitDtAssertions` with assert statements for 64 bit date and time ``LDT``

.. <legal notes>

legal notes
=================
| SPDX-FileCopyrightText: © 2022 ekvip automation GmbH <info@ekvip.de>
| SPDX-License-Identifier: Apache-2.0
| For details check: Apache-2.0_

.. _Apache-2.0: https://www.apache.org/licenses/LICENSE-2.0

.. </legal notes>

*)

PROPERTY dateAndTime :I64BitDtAssertions
GET
END_GET
END_PROPERTY

(*

short summary
=================
Returns the interface :ref:`I64BitDateAssertions` with assert statements for 64 bit date ``LDATE``

.. <legal notes>

legal notes
=================
| SPDX-FileCopyrightText: © 2022 ekvip automation GmbH <info@ekvip.de>
| SPDX-License-Identifier: Apache-2.0
| For details check: Apache-2.0_

.. _Apache-2.0: https://www.apache.org/licenses/LICENSE-2.0

.. </legal notes>

*)

PROPERTY dateOnly :I64BitDateAssertions
GET
END_GET
END_PROPERTY

(*

short summary
=================
Returns the interface :ref:`I64BitTodAssertions` with assert statements for 32 bit time of day ``LTOD``

.. <legal notes>

legal notes
=================
| SPDX-FileCopyrightText: © 2022 ekvip automation GmbH <info@ekvip.de>
| SPDX-License-Identifier: Apache-2.0
| For details check: Apache-2.0_

.. _Apache-2.0: https://www.apache.org/licenses/LICENSE-2.0

.. </legal notes>

*)

PROPERTY timeOfDay :I64BitTodAssertions
GET
END_GET
END_PROPERTY

END_INTERFACE

// ---- Assertor/Assertions/DateAndTimeAssertions/64Bit/LTOD/interfaces/I64BitTodAssertions.TcIO
(*

short summary
=================
This interface provides assert statements for 64 bit time of day ``LTOD``  

.. <legal notes>

legal notes
=================
| SPDX-FileCopyrightText: © 2022 ekvip automation GmbH <info@ekvip.de>
| SPDX-License-Identifier: Apache-2.0
| For details check: Apache-2.0_

.. _Apache-2.0: https://www.apache.org/licenses/LICENSE-2.0

.. </legal notes>

methods
==================

*)

INTERFACE I64BitTodAssertions EXTENDS __SYSTEM.IQueryInterface

(*

short summary
=================
This assertion method checks if the current value is equal to the expected value

.. <legal notes>

legal notes
=================
| SPDX-FileCopyrightText: © 2022 ekvip automation GmbH <info@ekvip.de>
| SPDX-License-Identifier: Apache-2.0
| For details check: Apache-2.0_

.. _Apache-2.0: https://www.apache.org/licenses/LICENSE-2.0

.. </legal notes>

parameters
=================

*)

METHOD valueIsEqualTo
VAR_INPUT
	(* current value to check *)
	currentValue	:LTOD;
	(* expected value to compare *)
	expectedValue	:LTOD;
	(* message if the assertion is false *)
	message			:AssertMessage;
END_VAR
END_METHOD

(*

short summary
=================
This assertion method checks if the current value is greater than the less value

.. <legal notes>

legal notes
=================
| SPDX-FileCopyrightText: © 2022 ekvip automation GmbH <info@ekvip.de>
| SPDX-License-Identifier: Apache-2.0
| For details check: Apache-2.0_

.. _Apache-2.0: https://www.apache.org/licenses/LICENSE-2.0

.. </legal notes>

parameters
=================

*)

METHOD valueIsGreaterThan
VAR_INPUT
	(* current value to check *)
	currentValue	:LTOD;
	(* less than lower limit *)
	lessValue		:LTOD;
	(* message if the assertion is false *)
	message			:AssertMessage;
END_VAR
END_METHOD

(*

short summary
=================
This assertion method checks if the current value is inside a limit

.. attention:: 
	limits are included: ``valueIsInRangeOf(ltod#3:0:0, ltod#3:0:0, ltod#3:0:0)`` is a true assertion

.. <legal notes>

legal notes
=================
| SPDX-FileCopyrightText: © 2022 ekvip automation GmbH <info@ekvip.de>
| SPDX-License-Identifier: Apache-2.0
| For details check: Apache-2.0_

.. _Apache-2.0: https://www.apache.org/licenses/LICENSE-2.0

.. </legal notes>

parameters
=================

*)

METHOD valueIsInRangeOf
VAR_INPUT
	(* lower limit for the current value *)
	lowerLimit		:LTOD;
	(* current value to check *)
	currentValue	:LTOD;
	(* upper limit for the current value *)
	upperLimit		:LTOD;
	(* message if the assertion is false *)
	message			:AssertMessage;
END_VAR
END_METHOD

(*

short summary
=================
This assertion method checks if the current value is less than the greater value

.. <legal notes>

legal notes
=================
| SPDX-FileCopyrightText: © 2022 ekvip automation GmbH <info@ekvip.de>
| SPDX-License-Identifier: Apache-2.0
| For details check: Apache-2.0_

.. _Apache-2.0: https://www.apache.org/licenses/LICENSE-2.0

.. </legal notes>

parameters
=================

*)

METHOD valueIsLessThan
VAR_INPUT
	(* current value to check *)
	currentValue	:LTOD;
	(* greater than upper limit *)
	greaterValue	:LTOD;
	(* message if the assertion is false *)
	message			:AssertMessage;
END_VAR
END_METHOD

(*

short summary
=================
This assertion method checks if the current value is less than or equal to the maximum value

.. <legal notes>

legal notes
=================
| SPDX-FileCopyrightText: © 2022 ekvip automation GmbH <info@ekvip.de>
| SPDX-License-Identifier: Apache-2.0
| For details check: Apache-2.0_

.. _Apache-2.0: https://www.apache.org/licenses/LICENSE-2.0

.. </legal notes>

parameters
=================

*)

METHOD valueIsMax
VAR_INPUT
	(* current value to check *)
	currentValue	:LTOD;
	(* upper limit for the current value *)
	maximumValue	:LTOD;
	(* message if the assertion is false *)
	message			:AssertMessage;
END_VAR
END_METHOD

(*

short summary
=================
This assertion method checks if the current value is greater than or equal to the minimum value

.. <legal notes>

legal notes
=================
| SPDX-FileCopyrightText: © 2022 ekvip automation GmbH <info@ekvip.de>
| SPDX-License-Identifier: Apache-2.0
| For details check: Apache-2.0_

.. _Apache-2.0: https://www.apache.org/licenses/LICENSE-2.0

.. </legal notes>

parameters
=================

*)

METHOD valueIsMin
VAR_INPUT
	(* current value to check *)
	currentValue	:LTOD;
	(* lower limit for the current value *)
	minimumValue	:LTOD;
	(* message if the assertion is false *)
	message			:AssertMessage;
END_VAR
END_METHOD

(*

short summary
=================
This assertion method checks if the current value is not equal to the unexpected value

.. <legal notes>

legal notes
=================
| SPDX-FileCopyrightText: © 2022 ekvip automation GmbH <info@ekvip.de>
| SPDX-License-Identifier: Apache-2.0
| For details check: Apache-2.0_

.. _Apache-2.0: https://www.apache.org/licenses/LICENSE-2.0

.. </legal notes>

parameters
=================

*)

METHOD valueIsNotEqualTo
VAR_INPUT
	(* current value to check *)
	currentValue	:LTOD;
	(* unexpected value to compare *)
	unexpectedValue	:LTOD;
	(* message if the assertion is false *)
	message			:AssertMessage;
END_VAR
END_METHOD

END_INTERFACE

// ---- Assertor/Assertions/DateAndTimeAssertions/interfaces/IDateAndTimeAssertions.TcIO
(*

short summary
=================
| This interface provides assert statements for date and time types
| For 32 bit date and time types use :ref:`IDateAndTimeAssertions.simple`

.. <legal notes>

legal notes
=================
| SPDX-FileCopyrightText: © 2022 ekvip automation GmbH <info@ekvip.de>
| SPDX-License-Identifier: Apache-2.0
| For details check: Apache-2.0_

.. _Apache-2.0: https://www.apache.org/licenses/LICENSE-2.0

.. </legal notes>

methods
==================

*)

INTERFACE IDateAndTimeAssertions EXTENDS __SYSTEM.IQueryInterface

(*

short summary
=================
Returns an interface with assert statements for 64 bit times 

.. <legal notes>

legal notes
=================
| SPDX-FileCopyrightText: © 2022 ekvip automation GmbH <info@ekvip.de>
| SPDX-License-Identifier: Apache-2.0
| For details check: Apache-2.0_

.. _Apache-2.0: https://www.apache.org/licenses/LICENSE-2.0

.. </legal notes>

*)

PROPERTY long :ILongDateAndTimeAssertions
GET
END_GET
END_PROPERTY

(*

short summary
=================
Returns the interface :ref:`ISimpleDateAndTimeAssertions` with assert statements for date and time types with 32 bit length

.. <legal notes>

legal notes
=================
| SPDX-FileCopyrightText: © 2022 ekvip automation GmbH <info@ekvip.de>
| SPDX-License-Identifier: Apache-2.0
| For details check: Apache-2.0_

.. _Apache-2.0: https://www.apache.org/licenses/LICENSE-2.0

.. </legal notes>

methods
==================

*)

PROPERTY simple :ISimpleDateAndTimeAssertions
GET
END_GET
END_PROPERTY

END_INTERFACE

// ---- Assertor/Assertions/FloatAssertions/interfaces/IFloatAssertions.TcIO
(*

short summary
=================
| This interface provides assert statements for floatings (``REAL`` and ``LREAL``)
| For 32 bit floats (``REAL``) use :ref:`IFloatAssertions.single`
| For 64 bit floats (``LREAL``) use :ref:`IFloatAssertions.double`

.. <legal notes>

legal notes
=================
| SPDX-FileCopyrightText: © 2022 ekvip automation GmbH <info@ekvip.de>
| SPDX-License-Identifier: Apache-2.0
| For details check: Apache-2.0_

.. _Apache-2.0: https://www.apache.org/licenses/LICENSE-2.0

.. </legal notes>

methods
==================

*)

INTERFACE IFloatAssertions EXTENDS __SYSTEM.IQueryInterface

(*

short summary
=================
Returns the interface :ref:`ILrealAssertions` with assert statements for 64 bit floatings (``LREAL``)

.. <legal notes>

legal notes
=================
| SPDX-FileCopyrightText: © 2022 ekvip automation GmbH <info@ekvip.de>
| SPDX-License-Identifier: Apache-2.0
| For details check: Apache-2.0_

.. _Apache-2.0: https://www.apache.org/licenses/LICENSE-2.0

.. </legal notes>

*)

PROPERTY double :ILrealAssertions
GET
END_GET
END_PROPERTY

(*

short summary
=================
Returns the interface :ref:`IRealAssertions` with assert statements for 32 bit floatings (``REAL``)

.. <legal notes>

legal notes
=================
| SPDX-FileCopyrightText: © 2022 ekvip automation GmbH <info@ekvip.de>
| SPDX-License-Identifier: Apache-2.0
| For details check: Apache-2.0_

.. _Apache-2.0: https://www.apache.org/licenses/LICENSE-2.0

.. </legal notes>

*)

PROPERTY single :IRealAssertions
GET
END_GET
END_PROPERTY

END_INTERFACE

// ---- Assertor/Assertions/FloatAssertions/Lreal/interfaces/ILrealAssertions.TcIO
(*

short summary
=================
This interface provides assert statements for 64 bit floatings (``LREAL``) 

.. <legal notes>

legal notes
=================
| SPDX-FileCopyrightText: © 2022 ekvip automation GmbH <info@ekvip.de>
| SPDX-License-Identifier: Apache-2.0
| For details check: Apache-2.0_

.. _Apache-2.0: https://www.apache.org/licenses/LICENSE-2.0

.. </legal notes>

methods
==================

*)

INTERFACE ILrealAssertions EXTENDS __SYSTEM.IQueryInterface

(*

short summary
=================
This assertion method checks if the current value is a number (NOT NaN)
for details check `IEEE 754`_

.. _IEEE 754: https://en.wikipedia.org/wiki/IEEE_754

.. <legal notes>

legal notes
=================
| SPDX-FileCopyrightText: © 2023 ekvip automation GmbH <info@ekvip.de>
| SPDX-License-Identifier: Apache-2.0
| For details check: Apache-2.0_

.. _Apache-2.0: https://www.apache.org/licenses/LICENSE-2.0

.. </legal notes>

parameters
=================

*)

METHOD valueIsANumber
VAR_INPUT
	(* current value to check *)
	currentValue	:LREAL;
	(* message if the assertion is false *)
	message			:AssertMessage;
END_VAR
END_METHOD

(*

short summary
=================
This assertion method checks if the current value is equal to the expected value

.. attention:: 
	Nothing is equal to NaN, that means if ``currentValue`` OR ``expectedValue`` OR ``tolerance``
	is NaN then is the assertion false. For details check `IEEE 754`_

.. attention:: 
	infinity is equal to infinity and -infinity is equal to -infinity, that means if
	``currentValue`` AND ``expectedValue`` have the value infinity 
	OR ``currentValue`` AND ``expectedValue`` have the value -infinity
	the assertion is TRUE. For details check `IEEE 754`_

.. attention:: 
	If ``tolerance`` has the value infinity or -infinity and 
	``currentValue`` is not NaN and ``expectedValue`` is not NaN
	then is the assertion true. For details check `IEEE 754`_

.. _IEEE 754: https://en.wikipedia.org/wiki/IEEE_754

.. <legal notes>

legal notes
=================
| SPDX-FileCopyrightText: © 2022 ekvip automation GmbH <info@ekvip.de>
| SPDX-License-Identifier: Apache-2.0
| For details check: Apache-2.0_

.. _Apache-2.0: https://www.apache.org/licenses/LICENSE-2.0

.. </legal notes>

parameters
=================

*)

METHOD valueIsEqualTo
VAR_INPUT
	(* current value to check *)
	currentValue	:LREAL;
	(* expected value to compare *)
	expectedValue	:LREAL;
	(* tolerance to compensate twiddling floats, it has no sign *)
	tolerance		:LREAL;
	(* message if the assertion is false *)
	message			:AssertMessage;
END_VAR
END_METHOD

(*

short summary
=================
This assertion method checks if the current value is finite
(NOT (infinty OR -inifinity)), for details check `IEEE 754`_

.. _IEEE 754: https://en.wikipedia.org/wiki/IEEE_754

.. <legal notes>

legal notes
=================
| SPDX-FileCopyrightText: © 2023 ekvip automation GmbH <info@ekvip.de>
| SPDX-License-Identifier: Apache-2.0
| For details check: Apache-2.0_

.. _Apache-2.0: https://www.apache.org/licenses/LICENSE-2.0

.. </legal notes>

parameters
=================

*)

METHOD valueIsFinite
VAR_INPUT
	(* current value to check *)
	currentValue	:LREAL;
	(* message if the assertion is false *)
	message			:AssertMessage;
END_VAR
END_METHOD

(*

short summary
=================
This assertion method checks if the current value is greater than the less value

.. attention:: 
	Any comparsion to NaN is ``FALSE`` that means if ``currentValue`` OR ``lessValue``
	is NaN then is the assertion false.
	For details check `IEEE 754`_ and the truth table below.

.. attention:: 
	Every number is smaller than infinity except -infinity, it's equal.
	Every number is greater than -infinity except -infinity, it's equal.
	For details check `IEEE 754`_ and the truth table below.

.. _IEEE 754: https://en.wikipedia.org/wiki/IEEE_754

truth table for special values
===============================
+----------------------+-------------------+---------------+
| **``currentValue``** | **``lessValue``** | **assertion** |
+======================+===================+===============+
| NaN                  | Any value         | FASLE         |
+----------------------+-------------------+---------------+
| Any value            | NaN               | FALSE         |
+----------------------+-------------------+---------------+
| infinity             | NOT NaN           | TRUE          |
|                      | NOT infinity      |               |
+----------------------+-------------------+---------------+
| -infinty             | Any value         | FALSE         |
+----------------------+-------------------+---------------+
| Any value            | infinity          | FALSE         |
+----------------------+-------------------+---------------+
| NOT NaN              | -inifinity        | TRUE          |
| NOT -infinity        |                   |               |
+----------------------+-------------------+---------------+

.. <legal notes>

legal notes
=================
| SPDX-FileCopyrightText: © 2022 ekvip automation GmbH <info@ekvip.de>
| SPDX-License-Identifier: Apache-2.0
| For details check: Apache-2.0_

.. _Apache-2.0: https://www.apache.org/licenses/LICENSE-2.0

.. </legal notes>

parameters
=================

*)

METHOD valueIsGreaterThan
VAR_INPUT
	(* current value to check *)
	currentValue	:LREAL;
	(* less than lower limit *)
	lessValue		:LREAL;
	(* message if the assertion is false *)
	message			:AssertMessage;
END_VAR
END_METHOD

(*

short summary
=================
This assertion method checks if the current value is infinite
(infinty OR -inifinity), for details check `IEEE 754`_

.. _IEEE 754: https://en.wikipedia.org/wiki/IEEE_754

.. <legal notes>

legal notes
=================
| SPDX-FileCopyrightText: © 2023 ekvip automation GmbH <info@ekvip.de>
| SPDX-License-Identifier: Apache-2.0
| For details check: Apache-2.0_

.. _Apache-2.0: https://www.apache.org/licenses/LICENSE-2.0

.. </legal notes>

parameters
=================

*)

METHOD valueIsInfinite
VAR_INPUT
	(* current value to check *)
	currentValue	:LREAL;
	(* message if the assertion is false *)
	message			:AssertMessage;
END_VAR
END_METHOD

(*

short summary
=================
This assertion method checks if the current value is inside a limit

.. attention:: 
	limits are included: ``valueIsInRangeOf(3.0, 3.0, 3.0)`` is a true assertion

.. attention:: 
	Any comparsion to NaN is ``FALSE`` that means 
	if ``lowerLimit`` OR ``currentValue`` OR ``upperLimit``
	is NaN then is the assertion false.
	For details check `IEEE 754`_ and the truth table below.

.. attention:: 
	Every number is smaller than infinity except -infinity, it's equal.
	Every number is greater than -infinity except -infinity, it's equal.
	For details check `IEEE 754`_ and the truth table below.

.. _IEEE 754: https://en.wikipedia.org/wiki/IEEE_754

truth table for special values
===============================
+--------------------+----------------------+--------------------+---------------+
| **``lowerLimit``** | **``currentValue``** | **``upperLimit``** | **assertion** |
+====================+======================+====================+===============+
| NaN                | Any value            | Any value          | FASLE         |
+--------------------+----------------------+--------------------+---------------+
| Any value          | NaN                  | Any value          | FALSE         |
+--------------------+----------------------+--------------------+---------------+
| Any value          | Any value            | NaN                | FALSE         |
+--------------------+----------------------+--------------------+---------------+
| -infinity          | NOT NaN              | infinity           | TRUE          |
+--------------------+----------------------+--------------------+---------------+
| infinity           | Any value            | -infinity          | FALSE         |
+--------------------+----------------------+--------------------+---------------+
| NOT -infinity      | -infinity            | Any value          | FALSE         |
+--------------------+----------------------+--------------------+---------------+
| Any value          | infinity             | NOT infinity       | FALSE         |
+--------------------+----------------------+--------------------+---------------+
| -infinity          | -infinity            | -infinity          | TRUE          |
+--------------------+----------------------+--------------------+---------------+
| infinity           | infinity             | infinity           | TRUE          |
+--------------------+----------------------+--------------------+---------------+
| -infinity          | NOT -infinity        | -infinity          | FALSE         |
+--------------------+----------------------+--------------------+---------------+
| infinity           | NOT infinity         | infinity           | FALSE         |
+--------------------+----------------------+--------------------+---------------+

.. <legal notes>

legal notes
=================
| SPDX-FileCopyrightText: © 2022 ekvip automation GmbH <info@ekvip.de>
| SPDX-License-Identifier: Apache-2.0
| For details check: Apache-2.0_

.. _Apache-2.0: https://www.apache.org/licenses/LICENSE-2.0

.. </legal notes>

parameters
=================

*)

METHOD valueIsInRangeOf
VAR_INPUT
	(* lower limit for the current value *)
	lowerLimit		:LREAL;
	(* current value to check *)
	currentValue	:LREAL;
	(* upper limit for the current value *)
	upperLimit		:LREAL;
	(* message if the assertion is false *)
	message			:AssertMessage;
END_VAR
END_METHOD

(*

short summary
=================
This assertion method checks if the current value is greater than the less value

.. attention::
	Any comparsion to NaN is ``FALSE`` that means if ``currentValue`` OR ``greaterValue``
	is NaN then is the assertion false.
	For details check `IEEE 754`_ and the truth table below.

.. attention::
	Every number is smaller than infinity except -infinity, it's equal.
	Every number is greater than -infinity except -infinity, it's equal.
	For details check `IEEE 754`_ and the truth table below.

.. _IEEE 754: https://en.wikipedia.org/wiki/IEEE_754

truth table for special values
===============================
+----------------------+----------------------+---------------+
| **``currentValue``** | **``greaterValue``** | **assertion** |
+======================+======================+===============+
| NaN                  | Any value            | FASLE         |
+----------------------+----------------------+---------------+
| Any value            | NaN                  | FALSE         |
+----------------------+----------------------+---------------+
| infinity             | Any value            | FALSE         |
+----------------------+----------------------+---------------+
| -infinty             | NOT NaN              | TRUE          |
|                      | NOT -infinity        |               |
+----------------------+----------------------+---------------+
| NOT NaN              | infinity             | TRUE          |
| NOT infinity         |                      |               |
+----------------------+----------------------+---------------+

.. <legal notes>

legal notes
=================
| SPDX-FileCopyrightText: © 2022 ekvip automation GmbH <info@ekvip.de>
| SPDX-License-Identifier: Apache-2.0
| For details check: Apache-2.0_

.. _Apache-2.0: https://www.apache.org/licenses/LICENSE-2.0

.. </legal notes>

parameters
=================

*)

METHOD valueIsLessThan
VAR_INPUT
	(* current value to check *)
	currentValue	:LREAL;
	(* greater than upper limit *)
	greaterValue	:LREAL;
	(* message if the assertion is false *)
	message			:AssertMessage;
END_VAR
END_METHOD

(*

short summary
=================
This assertion method checks if the current value is less than or equal to the maximum value

.. attention::
	Any comparsion to NaN is ``FALSE`` that means if ``currentValue`` OR ``maximumValue``
	is NaN then is the assertion false.
	For details check `IEEE 754`_ and the truth table below.

.. attention::
	Every number is smaller than infinity except -infinity, it's equal.
	Every number is greater than -infinity except -infinity, it's equal.
	For details check `IEEE 754`_ and the truth table below.

.. _IEEE 754: https://en.wikipedia.org/wiki/IEEE_754

truth table for special values
===============================
+----------------------+----------------------+---------------+
| **``currentValue``** | **``maximumValue``** | **assertion** |
+======================+======================+===============+
| NaN                  | Any value            | FASLE         |
+----------------------+----------------------+---------------+
| Any value            | NaN                  | FALSE         |
+----------------------+----------------------+---------------+
| NOT NaN              | infinity             | TRUE          |
+----------------------+----------------------+---------------+
| -infinity            | NOT NaN              | TRUE          |
+----------------------+----------------------+---------------+
| infinity             | NOT infinity         | FALSE         |
+----------------------+----------------------+---------------+
| NOT -infinity        | -infinity            | FALSE         |
+----------------------+----------------------+---------------+

.. <legal notes>

legal notes
=================
| SPDX-FileCopyrightText: © 2022 ekvip automation GmbH <info@ekvip.de>
| SPDX-License-Identifier: Apache-2.0
| For details check: Apache-2.0_

.. _Apache-2.0: https://www.apache.org/licenses/LICENSE-2.0

.. </legal notes>

parameters
=================

*)

METHOD valueIsMax
VAR_INPUT
	(* current value to check *)
	currentValue	:LREAL;
	(* upper limit for the current value *)
	maximumValue	:LREAL;
	(* message if the assertion is false *)
	message			:AssertMessage;
END_VAR
END_METHOD

(*

short summary
=================
This assertion method checks if the current value is greater than or equal to the minimum value

.. attention::
	Any comparsion to NaN is ``FALSE`` that means if ``currentValue`` OR ``minimumValue``
	is NaN then is the assertion false.
	For details check `IEEE 754`_ and the truth table below.

.. attention::
	Every number is smaller than infinity except -infinity, it's equal.
	Every number is greater than -infinity except -infinity, it's equal.
	For details check `IEEE 754`_ and the truth table below.

.. _IEEE 754: https://en.wikipedia.org/wiki/IEEE_754

truth table for special values
===============================
+----------------------+----------------------+---------------+
| **``currentValue``** | **``minimumValue``** | **assertion** |
+======================+======================+===============+
| NaN                  | Any value            | FASLE         |
+----------------------+----------------------+---------------+
| Any value            | NaN                  | FALSE         |
+----------------------+----------------------+---------------+
| infinity             | NOT NaN              | TRUE          |
+----------------------+----------------------+---------------+
| NOT NaN              | -infinity            | TRUE          |
+----------------------+----------------------+---------------+
| -infinity            | NOT -infinity        | FALSE         |
+----------------------+----------------------+---------------+
| NOT infinity         | infinity             | FALSE         |
+----------------------+----------------------+---------------+

.. <legal notes>

legal notes
=================
| SPDX-FileCopyrightText: © 2022 ekvip automation GmbH <info@ekvip.de>
| SPDX-License-Identifier: Apache-2.0
| For details check: Apache-2.0_

.. _Apache-2.0: https://www.apache.org/licenses/LICENSE-2.0

.. </legal notes>

parameters
=================

*)

METHOD valueIsMin
VAR_INPUT
	(* current value to check *)
	currentValue	:LREAL;
	(* lower limit for the current value *)
	minimumValue	:LREAL;
	(* message if the assertion is false *)
	message			:AssertMessage;
END_VAR
END_METHOD

(*

short summary
=================
This assertion method checks if the current value is a not a number (NaN)
for details check `IEEE 754`_

.. _IEEE 754: https://en.wikipedia.org/wiki/IEEE_754

.. <legal notes>

legal notes
=================
| SPDX-FileCopyrightText: © 2023 ekvip automation GmbH <info@ekvip.de>
| SPDX-License-Identifier: Apache-2.0
| For details check: Apache-2.0_

.. _Apache-2.0: https://www.apache.org/licenses/LICENSE-2.0

.. </legal notes>

parameters
=================

*)

METHOD valueIsNaN
VAR_INPUT
	(* current value to check *)
	currentValue	:LREAL;
	(* message if the assertion is false *)
	message			:AssertMessage;
END_VAR
END_METHOD

(*

short summary
=================
This assertion method checks if the current value is negative

.. attention::
	Any comparsion to NaN is ``FALSE`` that means if ``currentValue``
	is NaN then is the assertion false.
	For details check `IEEE 754`_.

.. attention::
	``currentValue`` has the value infinity means the assertion is false.
	``currentValue`` has the value -infinity means the assertion is true.
	``currentValue`` has the +0.0 means the assertion is false.
	``currentValue`` has the value -0.0 means the assertion is true.	
	For details check `IEEE 754`_.

.. _IEEE 754: https://en.wikipedia.org/wiki/IEEE_754

.. <legal notes>

legal notes
=================
| SPDX-FileCopyrightText: © 2022 ekvip automation GmbH <info@ekvip.de>
| SPDX-License-Identifier: Apache-2.0
| For details check: Apache-2.0_

.. _Apache-2.0: https://www.apache.org/licenses/LICENSE-2.0

.. </legal notes>

parameters
=================

*)

METHOD valueIsNegative
VAR_INPUT
	(* current value to check *)
	currentValue	:LREAL;
	(* message if the assertion is false *)
	message			:AssertMessage;
END_VAR
END_METHOD

(*

short summary
=================
This assertion method checks if the current value is negative infinite
(-infinty), for details check `IEEE 754`_

.. _IEEE 754: https://en.wikipedia.org/wiki/IEEE_754

.. <legal notes>

legal notes
=================
| SPDX-FileCopyrightText: © 2023 ekvip automation GmbH <info@ekvip.de>
| SPDX-License-Identifier: Apache-2.0
| For details check: Apache-2.0_

.. _Apache-2.0: https://www.apache.org/licenses/LICENSE-2.0

.. </legal notes>

parameters
=================

*)

METHOD valueIsNegativeInfinite
VAR_INPUT
	(* current value to check *)
	currentValue	:LREAL;
	(* message if the assertion is false *)
	message			:AssertMessage;
END_VAR
END_METHOD

(*

short summary
=================
This assertion method checks if the current value is +0.0
for details check `IEEE 754`_

.. _IEEE 754: https://en.wikipedia.org/wiki/IEEE_754

.. <legal notes>

legal notes
=================
| SPDX-FileCopyrightText: © 2023 ekvip automation GmbH <info@ekvip.de>
| SPDX-License-Identifier: Apache-2.0
| For details check: Apache-2.0_

.. _Apache-2.0: https://www.apache.org/licenses/LICENSE-2.0

.. </legal notes>

parameters
=================

*)

METHOD valueIsNegativeZero
VAR_INPUT
	(* current value to check *)
	currentValue	:LREAL;
	(* message if the assertion is false *)
	message			:AssertMessage;
END_VAR
END_METHOD

(*

short summary
=================
This assertion method checks if the current value is a normal number (not subnormal)
for details check `IEEE 754`_

.. _IEEE 754: https://en.wikipedia.org/wiki/IEEE_754

.. <legal notes>

legal notes
=================
| SPDX-FileCopyrightText: © 2023 ekvip automation GmbH <info@ekvip.de>
| SPDX-License-Identifier: Apache-2.0
| For details check: Apache-2.0_

.. _Apache-2.0: https://www.apache.org/licenses/LICENSE-2.0

.. </legal notes>

parameters
=================

*)

METHOD valueIsNormal
VAR_INPUT
	(* current value to check *)
	currentValue	:LREAL;
	(* message if the assertion is false *)
	message			:AssertMessage;
END_VAR
END_METHOD

(*

short summary
=================
This assertion method checks if the current value is not equal to the unexpected value

.. attention:: 
	Nothing is equal to NaN, that means if ``currentValue`` OR ``unexpectedValue`` OR ``tolerance``
	is NaN then is the assertion true. For details check `IEEE 754`_

.. attention:: 
	infinity is equal to infinity and -infinity is equal to -infinity, that means if
	``currentValue`` AND ``unexpectedValue`` have the value infinity 
	OR ``currentValue`` AND ``unexpectedValue`` have the value -infinity
	the assertion is false. For details check `IEEE 754`_

.. attention:: 
	If ``tolerance`` has the value infinity or -infinity and 
	``currentValue`` is not NaN and ``unexpectedValue`` is not NaN
	then is the assertion false. For details check `IEEE 754`_

.. _IEEE 754: https://en.wikipedia.org/wiki/IEEE_754

.. <legal notes>

legal notes
=================
| SPDX-FileCopyrightText: © 2022 ekvip automation GmbH <info@ekvip.de>
| SPDX-License-Identifier: Apache-2.0
| For details check: Apache-2.0_

.. _Apache-2.0: https://www.apache.org/licenses/LICENSE-2.0

.. </legal notes>

parameters
=================

*)

METHOD valueIsNotEqualTo
VAR_INPUT
	(* current value to check *)
	currentValue	:LREAL;
	(* unexpected value to compare *)
	unexpectedValue	:LREAL;
	(* tolerance to compensate twiddling floats, it has no sign *)
	tolerance		:LREAL;
	(* message if the assertion is false *)
	message			:AssertMessage;
END_VAR
END_METHOD

(*

short summary
=================
This assertion method checks if the current value is not negative infinite
NOT (-infinty), for details check `IEEE 754`_

.. _IEEE 754: https://en.wikipedia.org/wiki/IEEE_754

.. <legal notes>

legal notes
=================
| SPDX-FileCopyrightText: © 2023 ekvip automation GmbH <info@ekvip.de>
| SPDX-License-Identifier: Apache-2.0
| For details check: Apache-2.0_

.. _Apache-2.0: https://www.apache.org/licenses/LICENSE-2.0

.. </legal notes>

parameters
=================

*)

METHOD valueIsNotNegativeInfinite
VAR_INPUT
	(* current value to check *)
	currentValue	:LREAL;
	(* message if the assertion is false *)
	message			:AssertMessage;
END_VAR
END_METHOD

(*

short summary
=================
This assertion method checks if the current value is not positive infinite
NOT (infinty), for details check `IEEE 754`_

.. _IEEE 754: https://en.wikipedia.org/wiki/IEEE_754

.. <legal notes>

legal notes
=================
| SPDX-FileCopyrightText: © 2023 ekvip automation GmbH <info@ekvip.de>
| SPDX-License-Identifier: Apache-2.0
| For details check: Apache-2.0_

.. _Apache-2.0: https://www.apache.org/licenses/LICENSE-2.0

.. </legal notes>

parameters
=================

*)

METHOD valueIsNotPositiveInfinite
VAR_INPUT
	(* current value to check *)
	currentValue	:LREAL;
	(* message if the assertion is false *)
	message			:AssertMessage;
END_VAR
END_METHOD

(*

short summary
=================
This assertion method checks if the current value is a non special number
(NOT (NaN OR infinty OR -inifinity)), for details check `IEEE 754`_

.. _IEEE 754: https://en.wikipedia.org/wiki/IEEE_754

.. <legal notes>

legal notes
=================
| SPDX-FileCopyrightText: © 2023 ekvip automation GmbH <info@ekvip.de>
| SPDX-License-Identifier: Apache-2.0
| For details check: Apache-2.0_

.. _Apache-2.0: https://www.apache.org/licenses/LICENSE-2.0

.. </legal notes>

parameters
=================

*)

METHOD valueIsNotSpecial : BOOL
VAR_INPUT
	(* current value to check *)
	currentValue	:LREAL;
	(* message if the assertion is false *)
	message			:AssertMessage;
END_VAR
END_METHOD

(*

short summary
=================
This assertion method checks if the current value is positve

.. attention::
	Any comparsion to NaN is ``FALSE`` that means if ``currentValue``
	is NaN then is the assertion false.
	For details check `IEEE 754`_.

.. attention::
	``currentValue`` has the value infinity means the assertion is true.
	``currentValue`` has the value -infinity means the assertion is false.
	``currentValue`` has the +0.0 means the assertion is true.
	``currentValue`` has the value -0.0 means the assertion is false.	
	For details check `IEEE 754`_.

.. _IEEE 754: https://en.wikipedia.org/wiki/IEEE_754

.. <legal notes>

legal notes
=================
| SPDX-FileCopyrightText: © 2022 ekvip automation GmbH <info@ekvip.de>
| SPDX-License-Identifier: Apache-2.0
| For details check: Apache-2.0_

.. _Apache-2.0: https://www.apache.org/licenses/LICENSE-2.0

.. </legal notes>

parameters
=================

*)

METHOD valueIsPositive
VAR_INPUT
	(* current value to check *)
	currentValue	:LREAL;
	(* message if the assertion is false *)
	message			:AssertMessage;
END_VAR
END_METHOD

(*

short summary
=================
This assertion method checks if the current value is positive infinite
(infinty), for details check `IEEE 754`_

.. _IEEE 754: https://en.wikipedia.org/wiki/IEEE_754

.. <legal notes>

legal notes
=================
| SPDX-FileCopyrightText: © 2023 ekvip automation GmbH <info@ekvip.de>
| SPDX-License-Identifier: Apache-2.0
| For details check: Apache-2.0_

.. _Apache-2.0: https://www.apache.org/licenses/LICENSE-2.0

.. </legal notes>

parameters
=================

*)

METHOD valueIsPositiveInfinite
VAR_INPUT
	(* current value to check *)
	currentValue	:LREAL;
	(* message if the assertion is false *)
	message			:AssertMessage;
END_VAR
END_METHOD

(*

short summary
=================
This assertion method checks if the current value is -0.0
for details check `IEEE 754`_

.. _IEEE 754: https://en.wikipedia.org/wiki/IEEE_754

.. <legal notes>

legal notes
=================
| SPDX-FileCopyrightText: © 2023 ekvip automation GmbH <info@ekvip.de>
| SPDX-License-Identifier: Apache-2.0
| For details check: Apache-2.0_

.. _Apache-2.0: https://www.apache.org/licenses/LICENSE-2.0

.. </legal notes>

parameters
=================

*)

METHOD valueIsPositiveZero
VAR_INPUT
	(* current value to check *)
	currentValue	:LREAL;
	(* message if the assertion is false *)
	message			:AssertMessage;
END_VAR
END_METHOD

(*

short summary
=================
This assertion method checks if the current value is a special
(NaN OR infinty OR -inifinity), for details check `IEEE 754`_

.. _IEEE 754: https://en.wikipedia.org/wiki/IEEE_754

.. <legal notes>

legal notes
=================
| SPDX-FileCopyrightText: © 2023 ekvip automation GmbH <info@ekvip.de>
| SPDX-License-Identifier: Apache-2.0
| For details check: Apache-2.0_

.. _Apache-2.0: https://www.apache.org/licenses/LICENSE-2.0

.. </legal notes>

parameters
=================

*)

METHOD valueIsSpecial
VAR_INPUT
	(* current value to check *)
	currentValue	:LREAL;
	(* message if the assertion is false *)
	message			:AssertMessage;
END_VAR
END_METHOD

(*

short summary
=================
This assertion method checks if the current value is a subnormal number
for details check `IEEE 754`_

.. _IEEE 754: https://en.wikipedia.org/wiki/IEEE_754

.. <legal notes>

legal notes
=================
| SPDX-FileCopyrightText: © 2023 ekvip automation GmbH <info@ekvip.de>
| SPDX-License-Identifier: Apache-2.0
| For details check: Apache-2.0_

.. _Apache-2.0: https://www.apache.org/licenses/LICENSE-2.0

.. </legal notes>

parameters
=================

*)

METHOD valueIsSubnormal
VAR_INPUT
	(* current value to check *)
	currentValue	:LREAL;
	(* message if the assertion is false *)
	message			:AssertMessage;
END_VAR
END_METHOD

END_INTERFACE

// ---- Assertor/Assertions/FloatAssertions/Real/interfaces/IRealAssertions.TcIO
(*

short summary
=================
This interface provides assert statements for 32 bit floatings (``REAL``)

.. <legal notes>

legal notes
=================
| SPDX-FileCopyrightText: © 2022 ekvip automation GmbH <info@ekvip.de>
| SPDX-License-Identifier: Apache-2.0
| For details check: Apache-2.0_

.. _Apache-2.0: https://www.apache.org/licenses/LICENSE-2.0

.. </legal notes>

methods
==================

*)

INTERFACE IRealAssertions EXTENDS __SYSTEM.IQueryInterface

(*

short summary
=================
This assertion method checks if the current value is a number (NOT NaN)
for details check `IEEE 754`_

.. _IEEE 754: https://en.wikipedia.org/wiki/IEEE_754

.. <legal notes>

legal notes
=================
| SPDX-FileCopyrightText: © 2023 ekvip automation GmbH <info@ekvip.de>
| SPDX-License-Identifier: Apache-2.0
| For details check: Apache-2.0_

.. _Apache-2.0: https://www.apache.org/licenses/LICENSE-2.0

.. </legal notes>

parameters
=================

*)

METHOD valueIsANumber
VAR_INPUT
	(* current value to check *)
	currentValue	:REAL;
	(* message if the assertion is false *)
	message			:AssertMessage;
END_VAR
END_METHOD

(*

short summary
=================
This assertion method checks if the current value is equal to the expected value

.. attention:: 
	Nothing is equal to NaN, that means if ``currentValue`` OR ``expectedValue`` OR ``tolerance``
	is NaN then is the assertion false. For details check `IEEE 754`_

.. attention:: 
	infinity is equal to infinity and -infinity is equal to -infinity, that means if
	``currentValue`` AND ``expectedValue`` have the value infinity 
	OR ``currentValue`` AND ``expectedValue`` have the value -infinity
	the assertion is TRUE. For details check `IEEE 754`_

.. attention:: 
	If ``tolerance`` has the value infinity or -infinity and 
	``currentValue`` is not NaN and ``expectedValue`` is not NaN
	then is the assertion true. For details check `IEEE 754`_

.. _IEEE 754: https://en.wikipedia.org/wiki/IEEE_754

.. <legal notes>

legal notes
=================
| SPDX-FileCopyrightText: © 2022 ekvip automation GmbH <info@ekvip.de>
| SPDX-License-Identifier: Apache-2.0
| For details check: Apache-2.0_

.. _Apache-2.0: https://www.apache.org/licenses/LICENSE-2.0

.. </legal notes>

parameters
=================

*)

METHOD valueIsEqualTo
VAR_INPUT
	(* current value to check *)
	currentValue	:REAL;
	(* expected value to compare *)
	expectedValue	:REAL;
	(* tolerance to compensate twiddling floats *)
	tolerance		:REAL;
	(* message if the assertion is false *)
	message			:AssertMessage;
END_VAR
END_METHOD

(*

short summary
=================
This assertion method checks if the current value is finite
(NOT (infinty OR -inifinity)), for details check `IEEE 754`_

.. _IEEE 754: https://en.wikipedia.org/wiki/IEEE_754

.. <legal notes>

legal notes
=================
| SPDX-FileCopyrightText: © 2023 ekvip automation GmbH <info@ekvip.de>
| SPDX-License-Identifier: Apache-2.0
| For details check: Apache-2.0_

.. _Apache-2.0: https://www.apache.org/licenses/LICENSE-2.0

.. </legal notes>

parameters
=================

*)

METHOD valueIsFinite
VAR_INPUT
	(* current value to check *)
	currentValue	:REAL;
	(* message if the assertion is false *)
	message			:AssertMessage;
END_VAR
END_METHOD

(*

short summary
=================
This assertion method checks if the current value is greater than the less value

.. attention:: 
	Any comparsion to NaN is ``FALSE`` that means if ``currentValue`` OR ``lessValue``
	is NaN then is the assertion false.
	For details check `IEEE 754`_ and the truth table below.

.. attention:: 
	Every number is smaller than infinity except -infinity, it's equal.
	Every number is greater than -infinity except -infinity, it's equal.
	For details check `IEEE 754`_ and the truth table below.

.. _IEEE 754: https://en.wikipedia.org/wiki/IEEE_754

truth table for special values
===============================
+----------------------+-------------------+---------------+
| **``currentValue``** | **``lessValue``** | **assertion** |
+======================+===================+===============+
| NaN                  | Any value         | FASLE         |
+----------------------+-------------------+---------------+
| Any value            | NaN               | FALSE         |
+----------------------+-------------------+---------------+
| infinity             | NOT NaN           | TRUE          |
|                      | NOT infinity      |               |
+----------------------+-------------------+---------------+
| -infinty             | Any value         | FALSE         |
+----------------------+-------------------+---------------+
| Any value            | infinity          | FALSE         |
+----------------------+-------------------+---------------+
| NOT NaN              | -inifinity        | TRUE          |
| NOT -infinity        |                   |               |
+----------------------+-------------------+---------------+

.. <legal notes>

legal notes
=================
| SPDX-FileCopyrightText: © 2022 ekvip automation GmbH <info@ekvip.de>
| SPDX-License-Identifier: Apache-2.0
| For details check: Apache-2.0_

.. _Apache-2.0: https://www.apache.org/licenses/LICENSE-2.0

.. </legal notes>

parameters
=================

*)

METHOD valueIsGreaterThan
VAR_INPUT
	(* current value to check *)
	currentValue	:REAL;
	(* less than lower limit *)
	lessValue		:REAL;
	(* message if the assertion is false *)
	message			:AssertMessage;
END_VAR
END_METHOD

(*

short summary
=================
This assertion method checks if the current value is infinite
(infinty OR -inifinity), for details check `IEEE 754`_

.. _IEEE 754: https://en.wikipedia.org/wiki/IEEE_754

.. <legal notes>

legal notes
=================
| SPDX-FileCopyrightText: © 2023 ekvip automation GmbH <info@ekvip.de>
| SPDX-License-Identifier: Apache-2.0
| For details check: Apache-2.0_

.. _Apache-2.0: https://www.apache.org/licenses/LICENSE-2.0

.. </legal notes>

parameters
=================

*)

METHOD valueIsInfinite
VAR_INPUT
	(* current value to check *)
	currentValue	:REAL;
	(* message if the assertion is false *)
	message			:AssertMessage;
END_VAR
END_METHOD

(*

short summary
=================
This assertion method checks if the current value is inside a limit

.. attention:: 
	limits are included: ``valueIsInRangeOf(3.0, 3.0, 3.0)`` is a true assertion

.. attention:: 
	Any comparsion to NaN is ``FALSE`` that means 
	if ``lowerLimit`` OR ``currentValue`` OR ``upperLimit``
	is NaN then is the assertion false.
	For details check `IEEE 754`_ and the truth table below.

.. attention:: 
	Every number is smaller than infinity except -infinity, it's equal.
	Every number is greater than -infinity except -infinity, it's equal.
	For details check `IEEE 754`_ and the truth table below.

.. _IEEE 754: https://en.wikipedia.org/wiki/IEEE_754

truth table for special values
===============================
+--------------------+----------------------+--------------------+---------------+
| **``lowerLimit``** | **``currentValue``** | **``upperLimit``** | **assertion** |
+====================+======================+====================+===============+
| NaN                | Any value            | Any value          | FASLE         |
+--------------------+----------------------+--------------------+---------------+
| Any value          | NaN                  | Any value          | FALSE         |
+--------------------+----------------------+--------------------+---------------+
| Any value          | Any value            | NaN                | FALSE         |
+--------------------+----------------------+--------------------+---------------+
| -infinity          | NOT NaN              | infinity           | TRUE          |
+--------------------+----------------------+--------------------+---------------+
| infinity           | Any value            | -infinity          | FALSE         |
+--------------------+----------------------+--------------------+---------------+
| NOT -infinity      | -infinity            | Any value          | FALSE         |
+--------------------+----------------------+--------------------+---------------+
| Any value          | infinity             | NOT infinity       | FALSE         |
+--------------------+----------------------+--------------------+---------------+
| -infinity          | -infinity            | -infinity          | TRUE          |
+--------------------+----------------------+--------------------+---------------+
| infinity           | infinity             | infinity           | TRUE          |
+--------------------+----------------------+--------------------+---------------+
| -infinity          | NOT -infinity        | -infinity          | FALSE         |
+--------------------+----------------------+--------------------+---------------+
| infinity           | NOT infinity         | infinity           | FALSE         |
+--------------------+----------------------+--------------------+---------------+

.. <legal notes>

legal notes
=================
| SPDX-FileCopyrightText: © 2022 ekvip automation GmbH <info@ekvip.de>
| SPDX-License-Identifier: Apache-2.0
| For details check: Apache-2.0_

.. _Apache-2.0: https://www.apache.org/licenses/LICENSE-2.0

.. </legal notes>

parameters
=================

*)

METHOD valueIsInRangeOf
VAR_INPUT
	(* lower limit for the current value *)
	lowerLimit		:REAL;
	(* current value to check *)
	currentValue	:REAL;
	(* upper limit for the current value *)
	upperLimit		:REAL;
	(* message if the assertion is false *)
	message			:AssertMessage;
END_VAR
END_METHOD

(*

short summary
=================
This assertion method checks if the current value is greater than the less value

.. attention::
	Any comparsion to NaN is ``FALSE`` that means if ``currentValue`` OR ``greaterValue``
	is NaN then is the assertion false.
	For details check `IEEE 754`_ and the truth table below.

.. attention::
	Every number is smaller than infinity except -infinity, it's equal.
	Every number is greater than -infinity except -infinity, it's equal.
	For details check `IEEE 754`_ and the truth table below.

.. _IEEE 754: https://en.wikipedia.org/wiki/IEEE_754

truth table for special values
===============================
+----------------------+----------------------+---------------+
| **``currentValue``** | **``greaterValue``** | **assertion** |
+======================+======================+===============+
| NaN                  | Any value            | FASLE         |
+----------------------+----------------------+---------------+
| Any value            | NaN                  | FALSE         |
+----------------------+----------------------+---------------+
| infinity             | Any value            | FALSE         |
+----------------------+----------------------+---------------+
| -infinty             | NOT NaN              | TRUE          |
|                      | NOT -infinity        |               |
+----------------------+----------------------+---------------+
| NOT NaN              | infinity             | TRUE          |
| NOT infinity         |                      |               |
+----------------------+----------------------+---------------+

.. <legal notes>

legal notes
=================
| SPDX-FileCopyrightText: © 2022 ekvip automation GmbH <info@ekvip.de>
| SPDX-License-Identifier: Apache-2.0
| For details check: Apache-2.0_

.. _Apache-2.0: https://www.apache.org/licenses/LICENSE-2.0

.. </legal notes>

parameters
=================

*)

METHOD valueIsLessThan
VAR_INPUT
	(* current value to check *)
	currentValue	:REAL;
	(* greater than upper limit *)
	greaterValue	:REAL;
	(* message if the assertion is false *)
	message			:AssertMessage;
END_VAR
END_METHOD

(*

short summary
=================
This assertion method checks if the current value is less than or equal to the maximum value

.. attention::
	Any comparsion to NaN is ``FALSE`` that means if ``currentValue`` OR ``maximumValue``
	is NaN then is the assertion false.
	For details check `IEEE 754`_ and the truth table below.

.. attention::
	Every number is smaller than infinity except -infinity, it's equal.
	Every number is greater than -infinity except -infinity, it's equal.
	For details check `IEEE 754`_ and the truth table below.

.. _IEEE 754: https://en.wikipedia.org/wiki/IEEE_754

truth table for special values
===============================
+----------------------+----------------------+---------------+
| **``currentValue``** | **``maximumValue``** | **assertion** |
+======================+======================+===============+
| NaN                  | Any value            | FASLE         |
+----------------------+----------------------+---------------+
| Any value            | NaN                  | FALSE         |
+----------------------+----------------------+---------------+
| NOT NaN              | infinity             | TRUE          |
+----------------------+----------------------+---------------+
| -infinity            | NOT NaN              | TRUE          |
+----------------------+----------------------+---------------+
| infinity             | NOT infinity         | FALSE         |
+----------------------+----------------------+---------------+
| NOT -infinity        | -infinity            | FALSE         |
+----------------------+----------------------+---------------+

.. <legal notes>

legal notes
=================
| SPDX-FileCopyrightText: © 2022 ekvip automation GmbH <info@ekvip.de>
| SPDX-License-Identifier: Apache-2.0
| For details check: Apache-2.0_

.. _Apache-2.0: https://www.apache.org/licenses/LICENSE-2.0

.. </legal notes>

parameters
=================

*)

METHOD valueIsMax
VAR_INPUT
	(* current value to check *)
	currentValue	:REAL;
	(* upper limit for the current value *)
	maximumValue	:REAL;
	(* message if the assertion is false *)
	message			:AssertMessage;
END_VAR
END_METHOD

(*

short summary
=================
This assertion method checks if the current value is greater than or equal to the minimum value

.. attention::
	Any comparsion to NaN is ``FALSE`` that means if ``currentValue`` OR ``minimumValue``
	is NaN then is the assertion false.
	For details check `IEEE 754`_ and the truth table below.

.. attention::
	Every number is smaller than infinity except -infinity, it's equal.
	Every number is greater than -infinity except -infinity, it's equal.
	For details check `IEEE 754`_ and the truth table below.

.. _IEEE 754: https://en.wikipedia.org/wiki/IEEE_754

truth table for special values
===============================
+----------------------+----------------------+---------------+
| **``currentValue``** | **``minimumValue``** | **assertion** |
+======================+======================+===============+
| NaN                  | Any value            | FASLE         |
+----------------------+----------------------+---------------+
| Any value            | NaN                  | FALSE         |
+----------------------+----------------------+---------------+
| infinity             | NOT NaN              | TRUE          |
+----------------------+----------------------+---------------+
| NOT NaN              | -infinity            | TRUE          |
+----------------------+----------------------+---------------+
| -infinity            | NOT -infinity        | FALSE         |
+----------------------+----------------------+---------------+
| NOT infinity         | infinity             | FALSE         |
+----------------------+----------------------+---------------+

.. <legal notes>

